LIN {X 0,Y 367.219,Z 542.125,A -85,B 0,C 180,E1 -12876.018,E2 -12876.018} C_VEL
LIN {X 0,Y 366.921,Z 543.374,A -85,B 0,C 180,E1 -12876.247,E2 -12876.247} C_VEL
LIN {X 0,Y 365.149,Z 553.236,A -85,B 0,C 180,E1 -12878.302,E2 -12878.302} C_VEL
LIN {X 0,Y 363.652,Z 562.404,A -85,B 0,C 180,E1 -12880.582,E2 -12880.582} C_VEL
LIN {X 0,Y 362.474,Z 570.103,A -85,B 0,C 180,E1 -12882.886,E2 -12882.886} C_VEL
LIN {X 0,Y 361.538,Z 576.427,A -85,B 0,C 180,E1 -12885.216,E2 -12885.216} C_VEL
LIN {X 0,Y 360.968,Z 581.274,A -85,B 0,C 180,E1 -12887.439,E2 -12887.439} C_VEL
LIN {X 0,Y 360.588,Z 584.605,A -85,B 0,C 180,E1 -12889.352,E2 -12889.352} C_VEL
LIN {X 0,Y 360.218,Z 587.726,A -85,B 0,C 180,E1 -12891.761,E2 -12891.761} C_VEL
LIN {X 0,Y 360.039,Z 589.765,A -85,B 0,C 180,E1 -12894.202,E2 -12894.202} C_VEL
LIN {X 0,Y 360.038,Z 590.58,A -85,B 0,C 180,E1 -12896.679,E2 -12896.679} C_VEL
LIN {X 0,Y 360.098,Z 590.255,A -85,B 0,C 180,E1 -12899.206,E2 -12899.206} C_VEL
LIN {X 0,Y 360.219,Z 588.701,A -85,B 0,C 180,E1 -12901.79,E2 -12901.79} C_VEL
LIN {X 0,Y 360.383,Z 587.415,A -85,B 0,C 180,E1 -12903.098,E2 -12903.098} C_VEL
LIN {X 0,Y 360.836,Z 583.71,A -85,B 0,C 180,E1 -12905.756,E2 -12905.756} C_VEL
LIN {X 0,Y 361.537,Z 578.446,A -85,B 0,C 180,E1 -12908.468,E2 -12908.468} C_VEL
LIN {X 0,Y 362.453,Z 572.426,A -85,B 0,C 180,E1 -12910.868,E2 -12910.868} C_VEL
LIN {X 0,Y 363.696,Z 564.839,A -85,B 0,C 180,E1 -12913.315,E2 -12913.315} C_VEL
LIN {X 0,Y 365.109,Z 556.956,A -85,B 0,C 180,E1 -12915.417,E2 -12915.417} C_VEL
LIN {X 0,Y 366.958,Z 547.569,A -85,B 0,C 180,E1 -12917.508,E2 -12917.508} C_VEL
LIN {X 0,Y 369.193,Z 536.056,A -85,B 0,C 180,E1 -12919.666,E2 -12919.666} C_VEL
LIN {X 0,Y 371.386,Z 524.57,A -85,B 0,C 180,E1 -12921.48,E2 -12921.48} C_VEL
LIN {X 0,Y 373.724,Z 512.125,A -85,B 0,C 180,E1 -12923.14,E2 -12923.14} C_VEL
LIN {X 0,Y 376.004,Z 499.108,A -85,B 0,C 180,E1 -12924.589,E2 -12924.589} C_VEL
LIN {X 0,Y 378.24,Z 484.852,A -85,B 0,C 180,E1 -12925.921,E2 -12925.921} C_VEL
LIN {X 0,Y 380.349,Z 469.499,A -85,B 0,C 180,E1 -12927.097,E2 -12927.097} C_VEL
LIN {X 0,Y 382.181,Z 454.471,A -85,B 0,C 180,E1 -12928.018,E2 -12928.018} C_VEL
LIN {X 0,Y 383.744,Z 437.956,A -85,B 0,C 180,E1 -12928.798,E2 -12928.798} C_VEL
LIN {X 0,Y 384.867,Z 421.878,A -85,B 0,C 180,E1 -12929.343,E2 -12929.343} C_VEL
LIN {X 0,Y 385.749,Z 399.249,A -85,B 0,C 180,E1 -12929.848,E2 -12929.848} C_VEL
LIN {X 0,Y 390.453,Z 263.095,A -85,B 0,C 180,E1 -12932.539,E2 -12932.539} C_VEL
LIN {X 0,Y 382.124,Z 246.592,A -85,B 0,C 180,E1 -12933.936,E2 -12933.936} C_VEL
LIN {X 0,Y 375.065,Z 234.123,A -85,B 0,C 180,E1 -12935.165,E2 -12935.165} C_VEL
LIN {X 0,Y 367.961,Z 222.595,A -85,B 0,C 180,E1 -12936.463,E2 -12936.463} C_VEL
LIN {X 0,Y 365.004,Z 218.068,A -85,B 0,C 180,E1 -12937.021,E2 -12937.021} C_VEL
LIN {X 0,Y 362.52,Z 214.897,A -85,B 0,C 180,E1 -12937.487,E2 -12937.487} C_VEL
LIN {X 0,Y 362.058,Z 213.583,A -85,B 0,C 180,E1 -12937.607,E2 -12937.607} C_VEL
LIN {X 0,Y 361.885,Z 212.725,A -85,B 0,C 180,E1 -12937.821,E2 -12937.821} C_VEL
LIN {X 0,Y 361.961,Z 212.701,A -85,B 0,C 180,E1 -12941.9,E2 -12941.9} C_VEL
LIN {X 0,Y 361.966,Z 212.707,A -85,B 0,C 180,E1 -12945.379,E2 -12945.379} C_VEL
LIN {X 0,Y 361.973,Z 212.708,A -85,B 0,C 180,E1 -12948.804,E2 -12948.804} C_VEL
LIN {X 0,Y 362.119,Z 212.69,A -85,B 0,C 180,E1 -12952.191,E2 -12952.191} C_VEL
LIN {X 0,Y 362.116,Z 212.689,A -85,B 0,C 180,E1 -12954.431,E2 -12954.431} C_VEL
LIN {X 0,Y 362.28,Z 212.673,A -85,B 0,C 180,E1 -12957.776,E2 -12957.776} C_VEL
LIN {X 0,Y 362.406,Z 212.656,A -85,B 0,C 180,E1 -12959.999,E2 -12959.999} C_VEL
LIN {X 0,Y 362.281,Z 212.668,A -85,B 0,C 180,E1 -12962.223,E2 -12962.223} C_VEL
LIN {X 0,Y 362.148,Z 212.685,A -85,B 0,C 180,E1 -12966.686,E2 -12966.686} C_VEL
LIN {X 0,Y 362.001,Z 212.699,A -85,B 0,C 180,E1 -12970.062,E2 -12970.062} C_VEL
LIN {X 0,Y 362,Z 212.704,A -85,B 0,C 180,E1 -12973.898,E2 -12973.898} C_VEL
LIN {X 0,Y 361.929,Z 212.711,A -85,B 0,C 180,E1 -12976.934,E2 -12976.934} C_VEL
LIN {X 0,Y 361.885,Z 212.719,A -85,B 0,C 180,E1 -12980.46,E2 -12980.46} C_VEL
LIN {X 0,Y 361.896,Z 212.713,A -85,B 0,C 180,E1 -12984.112,E2 -12984.112} C_VEL
LIN {X 0,Y 361.943,Z 212.709,A -85,B 0,C 180,E1 -12986.72,E2 -12986.72} C_VEL
LIN {X 0,Y 361.866,Z 212.72,A -85,B 0,C 180,E1 -12990.328,E2 -12990.328} C_VEL
LIN {X 0,Y 361.855,Z 212.719,A -85,B 0,C 180,E1 -12994.28,E2 -12994.28} C_VEL
LIN {X 0,Y 361.864,Z 212.723,A -85,B 0,C 180,E1 -12997.222,E2 -12997.222} C_VEL
LIN {X 0,Y 361.831,Z 212.716,A -85,B 0,C 180,E1 -13000.753,E2 -13000.753} C_VEL
LIN {X 0,Y 361.817,Z 212.721,A -85,B 0,C 180,E1 -13004.368,E2 -13004.368} C_VEL
LIN {X 0,Y 361.851,Z 212.759,A -85,B 0,C 180,E1 -13006.761,E2 -13006.761} C_VEL
LIN {X 0,Y 367.533,Z 227.613,A -85,B 0,C 180,E1 -13010.242,E2 -13010.242} C_VEL
LIN {X 0,Y 376.424,Z 243.115,A -85,B 0,C 180,E1 -13011.885,E2 -13011.885} C_VEL
LIN {X 0,Y 383.341,Z 256.26,A -85,B 0,C 180,E1 -13013.092,E2 -13013.092} C_VEL
LIN {X 0,Y 389.462,Z 269.123,A -85,B 0,C 180,E1 -13014.13,E2 -13014.13} C_VEL
LIN {X 0,Y 390.227,Z 274.285,A -85,B 0,C 180,E1 -13014.34,E2 -13014.34} C_VEL
LIN {X 0,Y 384.653,Z 436.559,A -85,B 0,C 180,E1 -13017.573,E2 -13017.573} C_VEL
LIN {X 0,Y 383.367,Z 452.919,A -85,B 0,C 180,E1 -13018.076,E2 -13018.076} C_VEL
LIN {X 0,Y 381.787,Z 468.385,A -85,B 0,C 180,E1 -13018.741,E2 -13018.741} C_VEL
LIN {X 0,Y 380.071,Z 483.377,A -85,B 0,C 180,E1 -13019.587,E2 -13019.587} C_VEL
LIN {X 0,Y 377.947,Z 498.249,A -85,B 0,C 180,E1 -13020.628,E2 -13020.628} C_VEL
LIN {X 0,Y 375.867,Z 511.427,A -85,B 0,C 180,E1 -13021.761,E2 -13021.761} C_VEL
LIN {X 0,Y 373.487,Z 525.086,A -85,B 0,C 180,E1 -13023.151,E2 -13023.151} C_VEL
LIN {X 0,Y 371.05,Z 538.425,A -85,B 0,C 180,E1 -13024.773,E2 -13024.773} C_VEL
LIN {X 0,Y 368.668,Z 551.545,A -85,B 0,C 180,E1 -13026.697,E2 -13026.697} C_VEL
LIN {X 0,Y 366.53,Z 562.654,A -85,B 0,C 180,E1 -13028.633,E2 -13028.633} C_VEL
LIN {X 0,Y 364.626,Z 573.2,A -85,B 0,C 180,E1 -13030.812,E2 -13030.812} C_VEL
LIN {X 0,Y 363.1,Z 582.538,A -85,B 0,C 180,E1 -13033.12,E2 -13033.12} C_VEL
LIN {X 0,Y 361.972,Z 590.178,A -85,B 0,C 180,E1 -13035.378,E2 -13035.378} C_VEL
LIN {X 0,Y 361.188,Z 596.418,A -85,B 0,C 180,E1 -13037.639,E2 -13037.639} C_VEL
LIN {X 0,Y 360.622,Z 601.516,A -85,B 0,C 180,E1 -13039.896,E2 -13039.896} C_VEL
LIN {X 0,Y 360.448,Z 605.517,A -85,B 0,C 180,E1 -13042.153,E2 -13042.153} C_VEL
LIN {X 0,Y 360.321,Z 608.437,A -85,B 0,C 180,E1 -13044.401,E2 -13044.401} C_VEL
LIN {X 0,Y 360.27,Z 610.381,A -85,B 0,C 180,E1 -13046.642,E2 -13046.642} C_VEL
LIN {X 0,Y 360.318,Z 611.296,A -85,B 0,C 180,E1 -13048.88,E2 -13048.88} C_VEL
LIN {X 0,Y 360.32,Z 611.276,A -85,B 0,C 180,E1 -13051.115,E2 -13051.115} C_VEL
LIN {X 0,Y 360.269,Z 610.225,A -85,B 0,C 180,E1 -13053.352,E2 -13053.352} C_VEL
LIN {X 0,Y 360.373,Z 607.805,A -85,B 0,C 180,E1 -13055.959,E2 -13055.959} C_VEL
LIN {X 0,Y 360.444,Z 605.156,A -85,B 0,C 180,E1 -13057.842,E2 -13057.842} C_VEL
LIN {X 0,Y 360.616,Z 601.081,A -85,B 0,C 180,E1 -13060.099,E2 -13060.099} C_VEL
LIN {X 0,Y 361.38,Z 594.327,A -85,B 0,C 180,E1 -13062.92,E2 -13062.92} C_VEL
LIN {X 0,Y 362.424,Z 585.587,A -85,B 0,C 180,E1 -13065.749,E2 -13065.749} C_VEL
LIN {X 0,Y 363.753,Z 576.983,A -85,B 0,C 180,E1 -13068.003,E2 -13068.003} C_VEL
LIN {X 0,Y 365.114,Z 568.067,A -85,B 0,C 180,E1 -13069.975,E2 -13069.975} C_VEL
LIN {X 0,Y 366.921,Z 557.712,A -85,B 0,C 180,E1 -13071.928,E2 -13071.928} C_VEL
LIN {X 0,Y 368.887,Z 546.364,A -85,B 0,C 180,E1 -13073.746,E2 -13073.746} C_VEL
LIN {X 0,Y 370.776,Z 535.379,A -85,B 0,C 180,E1 -13075.241,E2 -13075.241} C_VEL
LIN {X 0,Y 372.93,Z 522.597,A -85,B 0,C 180,E1 -13076.735,E2 -13076.735} C_VEL
LIN {X 0,Y 375.092,Z 508.802,A -85,B 0,C 180,E1 -13078.087,E2 -13078.087} C_VEL
LIN {X 0,Y 377.203,Z 494.008,A -85,B 0,C 180,E1 -13079.276,E2 -13079.276} C_VEL
LIN {X 0,Y 379.094,Z 478.909,A -85,B 0,C 180,E1 -13080.263,E2 -13080.263} C_VEL
LIN {X 0,Y 380.72,Z 463.094,A -85,B 0,C 180,E1 -13081.08,E2 -13081.08} C_VEL
LIN {X 0,Y 382.112,Z 447.18,A -85,B 0,C 180,E1 -13081.686,E2 -13081.686} C_VEL
LIN {X 0,Y 383.114,Z 429.543,A -85,B 0,C 180,E1 -13082.135,E2 -13082.135} C_VEL
LIN {X 0,Y 387.859,Z 273.803,A -85,B 0,C 180,E1 -13085.17,E2 -13085.17} C_VEL
LIN {X 0,Y 386.671,Z 267.24,A -85,B 0,C 180,E1 -13085.435,E2 -13085.435} C_VEL
LIN {X 0,Y 376.6,Z 246.193,A -85,B 0,C 180,E1 -13086.955,E2 -13086.955} C_VEL
LIN {X 0,Y 367.525,Z 229.148,A -85,B 0,C 180,E1 -13088.37,E2 -13088.37} C_VEL
LIN {X 0,Y 363.515,Z 217.682,A -85,B 0,C 180,E1 -13090.639,E2 -13090.639} C_VEL
LIN {X 0,Y 361.829,Z 212.725,A -85,B 0,C 180,E1 -13091.693,E2 -13091.693} C_VEL
LIN {X 0,Y 361.801,Z 212.72,A -85,B 0,C 180,E1 -13095.63,E2 -13095.63} C_VEL
LIN {X 0,Y 361.849,Z 212.713,A -85,B 0,C 180,E1 -13099.235,E2 -13099.235} C_VEL
LIN {X 0,Y 361.844,Z 212.712,A -85,B 0,C 180,E1 -13102.98,E2 -13102.98} C_VEL
LIN {X 0,Y 361.832,Z 212.721,A -85,B 0,C 180,E1 -13106.629,E2 -13106.629} C_VEL
LIN {X 0,Y 361.837,Z 212.723,A -85,B 0,C 180,E1 -13109.669,E2 -13109.669} C_VEL
LIN {X 0,Y 361.925,Z 212.693,A -85,B 0,C 180,E1 -13113.473,E2 -13113.473} C_VEL
LIN {X 0,Y 361.88,Z 212.722,A -85,B 0,C 180,E1 -13117.145,E2 -13117.145} C_VEL
LIN {X 0,Y 361.903,Z 212.692,A -85,B 0,C 180,E1 -13120.724,E2 -13120.724} C_VEL
LIN {X 0,Y 361.916,Z 212.715,A -85,B 0,C 180,E1 -13124.225,E2 -13124.225} C_VEL
LIN {X 0,Y 361.969,Z 212.684,A -85,B 0,C 180,E1 -13126.527,E2 -13126.527} C_VEL
LIN {X 0,Y 362.005,Z 212.694,A -85,B 0,C 180,E1 -13129.938,E2 -13129.938} C_VEL
LIN {X 0,Y 362.138,Z 212.681,A -85,B 0,C 180,E1 -13133.314,E2 -13133.314} C_VEL
LIN {X 0,Y 362.251,Z 212.65,A -85,B 0,C 180,E1 -13137.777,E2 -13137.777} C_VEL
LIN {X 0,Y 362.398,Z 212.651,A -85,B 0,C 180,E1 -13140.001,E2 -13140.001} C_VEL
LIN {X 0,Y 362.251,Z 212.673,A -85,B 0,C 180,E1 -13142.224,E2 -13142.224} C_VEL
LIN {X 0,Y 362.132,Z 212.682,A -85,B 0,C 180,E1 -13146.687,E2 -13146.687} C_VEL
LIN {X 0,Y 362.001,Z 212.695,A -85,B 0,C 180,E1 -13150.063,E2 -13150.063} C_VEL
LIN {X 0,Y 361.969,Z 212.7,A -85,B 0,C 180,E1 -13153.9,E2 -13153.9} C_VEL
LIN {X 0,Y 361.94,Z 212.696,A -85,B 0,C 180,E1 -13157.941,E2 -13157.941} C_VEL
LIN {X 0,Y 361.866,Z 212.717,A -85,B 0,C 180,E1 -13161.655,E2 -13161.655} C_VEL
LIN {X 0,Y 361.903,Z 212.699,A -85,B 0,C 180,E1 -13165.293,E2 -13165.293} C_VEL
LIN {X 0,Y 361.889,Z 212.71,A -85,B 0,C 180,E1 -13167.781,E2 -13167.781} C_VEL
LIN {X 0,Y 361.824,Z 212.719,A -85,B 0,C 180,E1 -13171.288,E2 -13171.288} C_VEL
LIN {X 0,Y 361.832,Z 212.715,A -85,B 0,C 180,E1 -13174.284,E2 -13174.284} C_VEL
LIN {X 0,Y 361.842,Z 212.721,A -85,B 0,C 180,E1 -13177.226,E2 -13177.226} C_VEL
LIN {X 0,Y 361.816,Z 212.722,A -85,B 0,C 180,E1 -13180.758,E2 -13180.758} C_VEL
LIN {X 0,Y 361.799,Z 212.716,A -85,B 0,C 180,E1 -13184.372,E2 -13184.372} C_VEL
LIN {X 0,Y 361.818,Z 212.727,A -85,B 0,C 180,E1 -13187.572,E2 -13187.572} C_VEL
LIN {X 0,Y 361.82,Z 212.716,A -85,B 0,C 180,E1 -13190.984,E2 -13190.984} C_VEL
LIN {X 0,Y 361.863,Z 212.712,A -85,B 0,C 180,E1 -13194.659,E2 -13194.659} C_VEL
LIN {X 0,Y 361.829,Z 212.726,A -85,B 0,C 180,E1 -13198.374,E2 -13198.374} C_VEL
LIN {X 0,Y 361.858,Z 212.718,A -85,B 0,C 180,E1 -13200.956,E2 -13200.956} C_VEL
LIN {X 0,Y 361.877,Z 212.714,A -85,B 0,C 180,E1 -13204.71,E2 -13204.71} C_VEL
LIN {X 0,Y 361.851,Z 212.72,A -85,B 0,C 180,E1 -13208.348,E2 -13208.348} C_VEL
LIN {X 0,Y 361.918,Z 212.72,A -85,B 0,C 180,E1 -13212.088,E2 -13212.088} C_VEL
LIN {X 0,Y 361.981,Z 212.704,A -85,B 0,C 180,E1 -13216.115,E2 -13216.115} C_VEL
LIN {X 0,Y 361.956,Z 212.707,A -85,B 0,C 180,E1 -13218.055,E2 -13218.055} C_VEL
LIN {X 0,Y 362.948,Z 215.516,A -85,B 0,C 180,E1 -13218.254,E2 -13218.254} C_VEL
LIN {X 0,Y 364.51,Z 217.644,A -85,B 0,C 180,E1 -13218.491,E2 -13218.491} C_VEL
LIN {X 0,Y 373.334,Z 232.468,A -85,B 0,C 180,E1 -13219.859,E2 -13219.859} C_VEL
LIN {X 0,Y 381.122,Z 247.442,A -85,B 0,C 180,E1 -13221.038,E2 -13221.038} C_VEL
LIN {X 0,Y 387.956,Z 261.424,A -85,B 0,C 180,E1 -13222.048,E2 -13222.048} C_VEL
LIN {X 0,Y 383.102,Z 417.262,A -85,B 0,C 180,E1 -13225.103,E2 -13225.103} C_VEL
LIN {X 0,Y 382.07,Z 433.744,A -85,B 0,C 180,E1 -13225.618,E2 -13225.618} C_VEL
LIN {X 0,Y 380.73,Z 449.833,A -85,B 0,C 180,E1 -13226.328,E2 -13226.328} C_VEL
LIN {X 0,Y 379.108,Z 465.262,A -85,B 0,C 180,E1 -13227.213,E2 -13227.213} C_VEL
LIN {X 0,Y 377.356,Z 479.93,A -85,B 0,C 180,E1 -13228.268,E2 -13228.268} C_VEL
LIN {X 0,Y 375.115,Z 495.059,A -85,B 0,C 180,E1 -13229.6,E2 -13229.6} C_VEL
LIN {X 0,Y 372.931,Z 508.887,A -85,B 0,C 180,E1 -13231.082,E2 -13231.082} C_VEL
LIN {X 0,Y 370.628,Z 522.373,A -85,B 0,C 180,E1 -13232.811,E2 -13232.811} C_VEL
LIN {X 0,Y 368.554,Z 534.4,A -85,B 0,C 180,E1 -13234.651,E2 -13234.651} C_VEL
LIN {X 0,Y 366.921,Z 543.374,A -85,B 0,C 180,E1 -13236.247,E2 -13236.247} C_VEL
LIN {X 0,Y 365.622,Z 547.103,A -85,B 0,C 180,E1 -13236.936,E2 -13236.936} C_VEL
LIN {X 0,Y 358.662,Z 557.399,A -85,B 0,C 180,E1 -13238.972,E2 -13238.972} C_VEL
LIN {X 0,Y 357.128,Z 560.591,A -85,B 0,C 180,E1 -13239.732,E2 -13239.732} C_VEL
LIN {X 0,Y 356.889,Z 561.583,A -85,B 0,C 180,E1 -13239.999,E2 -13239.999} C_VEL
LIN {X 0,Y 355.521,Z 570.101,A -85,B 0,C 180,E1 -13242.562,E2 -13242.562} C_VEL
LIN {X 0,Y 354.542,Z 576.449,A -85,B 0,C 180,E1 -13244.936,E2 -13244.936} C_VEL
LIN {X 0,Y 353.873,Z 582.045,A -85,B 0,C 180,E1 -13247.579,E2 -13247.579} C_VEL
LIN {X 0,Y 353.444,Z 585.626,A -85,B 0,C 180,E1 -13249.759,E2 -13249.759} C_VEL
LIN {X 0,Y 353.06,Z 588.471,A -85,B 0,C 180,E1 -13252.225,E2 -13252.225} C_VEL
LIN {X 0,Y 352.933,Z 590.215,A -85,B 0,C 180,E1 -13254.721,E2 -13254.721} C_VEL
LIN {X 0,Y 352.947,Z 590.86,A -85,B 0,C 180,E1 -13257.259,E2 -13257.259} C_VEL
LIN {X 0,Y 353.01,Z 590.23,A -85,B 0,C 180,E1 -13259.851,E2 -13259.851} C_VEL
LIN {X 0,Y 353.196,Z 588.343,A -85,B 0,C 180,E1 -13262.499,E2 -13262.499} C_VEL
LIN {X 0,Y 353.378,Z 586.897,A -85,B 0,C 180,E1 -13263.841,E2 -13263.841} C_VEL
LIN {X 0,Y 353.93,Z 582.903,A -85,B 0,C 180,E1 -13266.565,E2 -13266.565} C_VEL
LIN {X 0,Y 354.518,Z 578.826,A -85,B 0,C 180,E1 -13268.644,E2 -13268.644} C_VEL
LIN {X 0,Y 355.613,Z 572.211,A -85,B 0,C 180,E1 -13271.322,E2 -13271.322} C_VEL
LIN {X 0,Y 357.004,Z 564.09,A -85,B 0,C 180,E1 -13273.939,E2 -13273.939} C_VEL
LIN {X 0,Y 358.628,Z 556.076,A -85,B 0,C 180,E1 -13276.071,E2 -13276.071} C_VEL
LIN {X 0,Y 360.56,Z 546.533,A -85,B 0,C 180,E1 -13278.197,E2 -13278.197} C_VEL
LIN {X 0,Y 362.805,Z 535.508,A -85,B 0,C 180,E1 -13280.263,E2 -13280.263} C_VEL
LIN {X 0,Y 365.158,Z 523.855,A -85,B 0,C 180,E1 -13282.103,E2 -13282.103} C_VEL
LIN {X 0,Y 367.605,Z 511.217,A -85,B 0,C 180,E1 -13283.79,E2 -13283.79} C_VEL
LIN {X 0,Y 369.972,Z 498.095,A -85,B 0,C 180,E1 -13285.257,E2 -13285.257} C_VEL
LIN {X 0,Y 372.295,Z 483.968,A -85,B 0,C 180,E1 -13286.569,E2 -13286.569} C_VEL
LIN {X 0,Y 374.312,Z 469.787,A -85,B 0,C 180,E1 -13287.664,E2 -13287.664} C_VEL
LIN {X 0,Y 376.249,Z 454.47,A -85,B 0,C 180,E1 -13288.613,E2 -13288.613} C_VEL
LIN {X 0,Y 377.877,Z 437.865,A -85,B 0,C 180,E1 -13289.407,E2 -13289.407} C_VEL
LIN {X 0,Y 379.012,Z 422.225,A -85,B 0,C 180,E1 -13289.94,E2 -13289.94} C_VEL
LIN {X 0,Y 379.946,Z 399.352,A -85,B 0,C 180,E1 -13290.458,E2 -13290.458} C_VEL
LIN {X 0,Y 384.734,Z 265.474,A -85,B 0,C 180,E1 -13293.148,E2 -13293.148} C_VEL
LIN {X 0,Y 377.424,Z 250.859,A -85,B 0,C 180,E1 -13294.421,E2 -13294.421} C_VEL
LIN {X 0,Y 370.711,Z 238.798,A -85,B 0,C 180,E1 -13295.635,E2 -13295.635} C_VEL
LIN {X 0,Y 363.511,Z 227.092,A -85,B 0,C 180,E1 -13296.989,E2 -13296.989} C_VEL
LIN {X 0,Y 360.024,Z 222.128,A -85,B 0,C 180,E1 -13297.663,E2 -13297.663} C_VEL
LIN {X 0,Y 357.91,Z 218.725,A -85,B 0,C 180,E1 -13298.093,E2 -13298.093} C_VEL
LIN {X 0,Y 355.666,Z 216.157,A -85,B 0,C 180,E1 -13298.532,E2 -13298.532} C_VEL
LIN {X 0,Y 354.871,Z 213.682,A -85,B 0,C 180,E1 -13298.786,E2 -13298.786} C_VEL
LIN {X 0,Y 354.903,Z 213.577,A -85,B 0,C 180,E1 -13302.719,E2 -13302.719} C_VEL
LIN {X 0,Y 354.955,Z 213.585,A -85,B 0,C 180,E1 -13306.255,E2 -13306.255} C_VEL
LIN {X 0,Y 354.96,Z 213.58,A -85,B 0,C 180,E1 -13309.735,E2 -13309.735} C_VEL
LIN {X 0,Y 355.127,Z 213.563,A -85,B 0,C 180,E1 -13313.18,E2 -13313.18} C_VEL
LIN {X 0,Y 355.244,Z 213.549,A -85,B 0,C 180,E1 -13317.732,E2 -13317.732} C_VEL
LIN {X 0,Y 355.356,Z 213.534,A -85,B 0,C 180,E1 -13319.999,E2 -13319.999} C_VEL
LIN {X 0,Y 355.244,Z 213.544,A -85,B 0,C 180,E1 -13322.267,E2 -13322.267} C_VEL
LIN {X 0,Y 355.112,Z 213.561,A -85,B 0,C 180,E1 -13326.819,E2 -13326.819} C_VEL
LIN {X 0,Y 354.957,Z 213.576,A -85,B 0,C 180,E1 -13330.264,E2 -13330.264} C_VEL
LIN {X 0,Y 354.945,Z 213.584,A -85,B 0,C 180,E1 -13334.018,E2 -13334.018} C_VEL
LIN {X 0,Y 354.892,Z 213.588,A -85,B 0,C 180,E1 -13338.091,E2 -13338.091} C_VEL
LIN {X 0,Y 354.819,Z 213.595,A -85,B 0,C 180,E1 -13342.106,E2 -13342.106} C_VEL
LIN {X 0,Y 354.9,Z 213.59,A -85,B 0,C 180,E1 -13345.827,E2 -13345.827} C_VEL
LIN {X 0,Y 354.816,Z 213.596,A -85,B 0,C 180,E1 -13349.681,E2 -13349.681} C_VEL
LIN {X 0,Y 354.809,Z 213.599,A -85,B 0,C 180,E1 -13353.701,E2 -13353.701} C_VEL
LIN {X 0,Y 354.798,Z 213.599,A -85,B 0,C 180,E1 -13356.459,E2 -13356.459} C_VEL
LIN {X 0,Y 354.827,Z 213.601,A -85,B 0,C 180,E1 -13359.423,E2 -13359.423} C_VEL
LIN {X 0,Y 354.788,Z 213.606,A -85,B 0,C 180,E1 -13362.866,E2 -13362.866} C_VEL
LIN {X 0,Y 354.791,Z 213.658,A -85,B 0,C 180,E1 -13365.749,E2 -13365.749} C_VEL
LIN {X 0,Y 360.099,Z 227.361,A -85,B 0,C 180,E1 -13369.136,E2 -13369.136} C_VEL
LIN {X 0,Y 368.027,Z 240.648,A -85,B 0,C 180,E1 -13370.678,E2 -13370.678} C_VEL
LIN {X 0,Y 376.256,Z 255.76,A -85,B 0,C 180,E1 -13372.192,E2 -13372.192} C_VEL
LIN {X 0,Y 384.055,Z 271.958,A -85,B 0,C 180,E1 -13373.567,E2 -13373.567} C_VEL
LIN {X 0,Y 384.577,Z 275.959,A -85,B 0,C 180,E1 -13373.727,E2 -13373.727} C_VEL
LIN {X 0,Y 378.828,Z 436.068,A -85,B 0,C 180,E1 -13376.962,E2 -13376.962} C_VEL
LIN {X 0,Y 377.476,Z 452.712,A -85,B 0,C 180,E1 -13377.478,E2 -13377.478} C_VEL
LIN {X 0,Y 375.753,Z 468.781,A -85,B 0,C 180,E1 -13378.181,E2 -13378.181} C_VEL
LIN {X 0,Y 373.685,Z 485.569,A -85,B 0,C 180,E1 -13379.168,E2 -13379.168} C_VEL
LIN {X 0,Y 371.507,Z 500.008,A -85,B 0,C 180,E1 -13380.224,E2 -13380.224} C_VEL
LIN {X 0,Y 368.991,Z 514.956,A -85,B 0,C 180,E1 -13381.563,E2 -13381.563} C_VEL
LIN {X 0,Y 366.447,Z 528.64,A -85,B 0,C 180,E1 -13383.056,E2 -13383.056} C_VEL
LIN {X 0,Y 364.19,Z 540.37,A -85,B 0,C 180,E1 -13384.57,E2 -13384.57} C_VEL
LIN {X 0,Y 362.077,Z 551.511,A -85,B 0,C 180,E1 -13386.247,E2 -13386.247} C_VEL
LIN {X 0,Y 359.836,Z 562.578,A -85,B 0,C 180,E1 -13388.215,E2 -13388.215} C_VEL
LIN {X 0,Y 358.024,Z 572.093,A -85,B 0,C 180,E1 -13390.205,E2 -13390.205} C_VEL
LIN {X 0,Y 356.415,Z 581.386,A -85,B 0,C 180,E1 -13392.498,E2 -13392.498} C_VEL
LIN {X 0,Y 355.004,Z 590.035,A -85,B 0,C 180,E1 -13395.084,E2 -13395.084} C_VEL
LIN {X 0,Y 354.184,Z 596.269,A -85,B 0,C 180,E1 -13397.39,E2 -13397.39} C_VEL
LIN {X 0,Y 353.569,Z 601.352,A -85,B 0,C 180,E1 -13399.692,E2 -13399.692} C_VEL
LIN {X 0,Y 353.359,Z 605.343,A -85,B 0,C 180,E1 -13401.995,E2 -13401.995} C_VEL
LIN {X 0,Y 353.239,Z 608.25,A -85,B 0,C 180,E1 -13404.288,E2 -13404.288} C_VEL
LIN {X 0,Y 353.191,Z 610.19,A -85,B 0,C 180,E1 -13406.575,E2 -13406.575} C_VEL
LIN {X 0,Y 353.218,Z 611.093,A -85,B 0,C 180,E1 -13408.857,E2 -13408.857} C_VEL
LIN {X 0,Y 353.221,Z 611.068,A -85,B 0,C 180,E1 -13411.137,E2 -13411.137} C_VEL
LIN {X 0,Y 353.19,Z 610.004,A -85,B 0,C 180,E1 -13413.419,E2 -13413.419} C_VEL
LIN {X 0,Y 353.272,Z 607.792,A -85,B 0,C 180,E1 -13415.905,E2 -13415.905} C_VEL
LIN {X 0,Y 353.355,Z 604.913,A -85,B 0,C 180,E1 -13418,E2 -13418} C_VEL
LIN {X 0,Y 353.553,Z 600.825,A -85,B 0,C 180,E1 -13420.303,E2 -13420.303} C_VEL
LIN {X 0,Y 354.361,Z 594.051,A -85,B 0,C 180,E1 -13423.181,E2 -13423.181} C_VEL
LIN {X 0,Y 355.182,Z 587.17,A -85,B 0,C 180,E1 -13425.49,E2 -13425.49} C_VEL
LIN {X 0,Y 356.523,Z 578.922,A -85,B 0,C 180,E1 -13427.787,E2 -13427.787} C_VEL
LIN {X 0,Y 357.864,Z 570.444,A -85,B 0,C 180,E1 -13429.798,E2 -13429.798} C_VEL
LIN {X 0,Y 359.656,Z 560.442,A -85,B 0,C 180,E1 -13431.791,E2 -13431.791} C_VEL
LIN {X 0,Y 361.794,Z 548.753,A -85,B 0,C 180,E1 -13433.767,E2 -13433.767} C_VEL
LIN {X 0,Y 363.847,Z 537.071,A -85,B 0,C 180,E1 -13435.449,E2 -13435.449} C_VEL
LIN {X 0,Y 366.287,Z 523.374,A -85,B 0,C 180,E1 -13437.105,E2 -13437.105} C_VEL
LIN {X 0,Y 368.522,Z 509.751,A -85,B 0,C 180,E1 -13438.47,E2 -13438.47} C_VEL
LIN {X 0,Y 370.698,Z 495.143,A -85,B 0,C 180,E1 -13439.685,E2 -13439.685} C_VEL
LIN {X 0,Y 372.787,Z 479.278,A -85,B 0,C 180,E1 -13440.751,E2 -13440.751} C_VEL
LIN {X 0,Y 374.471,Z 463.663,A -85,B 0,C 180,E1 -13441.579,E2 -13441.579} C_VEL
LIN {X 0,Y 375.974,Z 446.995,A -85,B 0,C 180,E1 -13442.226,E2 -13442.226} C_VEL
LIN {X 0,Y 377.008,Z 429.378,A -85,B 0,C 180,E1 -13442.681,E2 -13442.681} C_VEL
LIN {X 0,Y 381.873,Z 274.132,A -85,B 0,C 180,E1 -13445.757,E2 -13445.757} C_VEL
LIN {X 0,Y 381.018,Z 270.109,A -85,B 0,C 180,E1 -13445.936,E2 -13445.936} C_VEL
LIN {X 0,Y 371.199,Z 249.636,A -85,B 0,C 180,E1 -13447.455,E2 -13447.455} C_VEL
LIN {X 0,Y 361.504,Z 231.441,A -85,B 0,C 180,E1 -13449.007,E2 -13449.007} C_VEL
LIN {X 0,Y 360.206,Z 228.75,A -85,B 0,C 180,E1 -13449.255,E2 -13449.255} C_VEL
LIN {X 0,Y 354.794,Z 213.594,A -85,B 0,C 180,E1 -13452.43,E2 -13452.43} C_VEL
LIN {X 0,Y 354.754,Z 213.599,A -85,B 0,C 180,E1 -13456.102,E2 -13456.102} C_VEL
LIN {X 0,Y 354.801,Z 213.591,A -85,B 0,C 180,E1 -13459.182,E2 -13459.182} C_VEL
LIN {X 0,Y 354.785,Z 213.596,A -85,B 0,C 180,E1 -13462.4,E2 -13462.4} C_VEL
LIN {X 0,Y 354.787,Z 213.6,A -85,B 0,C 180,E1 -13464.939,E2 -13464.939} C_VEL
LIN {X 0,Y 354.766,Z 213.587,A -85,B 0,C 180,E1 -13468.403,E2 -13468.403} C_VEL
LIN {X 0,Y 354.819,Z 213.598,A -85,B 0,C 180,E1 -13471.617,E2 -13471.617} C_VEL
LIN {X 0,Y 354.871,Z 213.572,A -85,B 0,C 180,E1 -13474.171,E2 -13474.171} C_VEL
LIN {X 0,Y 354.825,Z 213.596,A -85,B 0,C 180,E1 -13477.894,E2 -13477.894} C_VEL
LIN {X 0,Y 354.894,Z 213.58,A -85,B 0,C 180,E1 -13481.89,E2 -13481.89} C_VEL
LIN {X 0,Y 354.913,Z 213.573,A -85,B 0,C 180,E1 -13485.981,E2 -13485.981} C_VEL
LIN {X 0,Y 354.952,Z 213.572,A -85,B 0,C 180,E1 -13489.736,E2 -13489.736} C_VEL
LIN {X 0,Y 355.101,Z 213.558,A -85,B 0,C 180,E1 -13493.181,E2 -13493.181} C_VEL
LIN {X 0,Y 355.215,Z 213.524,A -85,B 0,C 180,E1 -13497.733,E2 -13497.733} C_VEL
LIN {X 0,Y 355.367,Z 213.527,A -85,B 0,C 180,E1 -13500.001,E2 -13500.001} C_VEL
LIN {X 0,Y 355.214,Z 213.548,A -85,B 0,C 180,E1 -13502.268,E2 -13502.268} C_VEL
LIN {X 0,Y 355.096,Z 213.56,A -85,B 0,C 180,E1 -13506.821,E2 -13506.821} C_VEL
LIN {X 0,Y 354.948,Z 213.569,A -85,B 0,C 180,E1 -13510.266,E2 -13510.266} C_VEL
LIN {X 0,Y 354.914,Z 213.58,A -85,B 0,C 180,E1 -13514.02,E2 -13514.02} C_VEL
LIN {X 0,Y 354.895,Z 213.571,A -85,B 0,C 180,E1 -13518.11,E2 -13518.11} C_VEL
LIN {X 0,Y 354.808,Z 213.599,A -85,B 0,C 180,E1 -13522.108,E2 -13522.108} C_VEL
LIN {X 0,Y 354.874,Z 213.571,A -85,B 0,C 180,E1 -13525.83,E2 -13525.83} C_VEL
LIN {X 0,Y 354.831,Z 213.597,A -85,B 0,C 180,E1 -13529.681,E2 -13529.681} C_VEL
LIN {X 0,Y 354.785,Z 213.587,A -85,B 0,C 180,E1 -13533.705,E2 -13533.705} C_VEL
LIN {X 0,Y 354.777,Z 213.605,A -85,B 0,C 180,E1 -13536.463,E2 -13536.463} C_VEL
LIN {X 0,Y 354.806,Z 213.58,A -85,B 0,C 180,E1 -13539.427,E2 -13539.427} C_VEL
LIN {X 0,Y 354.771,Z 213.604,A -85,B 0,C 180,E1 -13542.871,E2 -13542.871} C_VEL
LIN {X 0,Y 354.75,Z 213.595,A -85,B 0,C 180,E1 -13546.107,E2 -13546.107} C_VEL
LIN {X 0,Y 354.769,Z 213.601,A -85,B 0,C 180,E1 -13549.182,E2 -13549.182} C_VEL
LIN {X 0,Y 354.79,Z 213.604,A -85,B 0,C 180,E1 -13552.407,E2 -13552.407} C_VEL
LIN {X 0,Y 354.801,Z 213.59,A -85,B 0,C 180,E1 -13554.944,E2 -13554.944} C_VEL
LIN {X 0,Y 354.784,Z 213.603,A -85,B 0,C 180,E1 -13558.409,E2 -13558.409} C_VEL
LIN {X 0,Y 354.794,Z 213.601,A -85,B 0,C 180,E1 -13561.618,E2 -13561.618} C_VEL
LIN {X 0,Y 354.829,Z 213.598,A -85,B 0,C 180,E1 -13565.661,E2 -13565.661} C_VEL
LIN {X 0,Y 354.823,Z 213.6,A -85,B 0,C 180,E1 -13569.117,E2 -13569.117} C_VEL
LIN {X 0,Y 354.858,Z 213.596,A -85,B 0,C 180,E1 -13572.721,E2 -13572.721} C_VEL
LIN {X 0,Y 354.94,Z 213.581,A -85,B 0,C 180,E1 -13576.258,E2 -13576.258} C_VEL
LIN {X 0,Y 354.961,Z 213.76,A -85,B 0,C 180,E1 -13577.242,E2 -13577.242} C_VEL
LIN {X 0,Y 355.953,Z 216.498,A -85,B 0,C 180,E1 -13577.437,E2 -13577.437} C_VEL
LIN {X 0,Y 357.579,Z 218.773,A -85,B 0,C 180,E1 -13577.695,E2 -13577.695} C_VEL
LIN {X 0,Y 367.054,Z 234.219,A -85,B 0,C 180,E1 -13579.2,E2 -13579.2} C_VEL
LIN {X 0,Y 375.712,Z 250.759,A -85,B 0,C 180,E1 -13580.553,E2 -13580.553} C_VEL
LIN {X 0,Y 381.978,Z 263.827,A -85,B 0,C 180,E1 -13581.505,E2 -13581.505} C_VEL
LIN {X 0,Y 376.992,Z 417.214,A -85,B 0,C 180,E1 -13584.554,E2 -13584.554} C_VEL
LIN {X 0,Y 375.948,Z 433.742,A -85,B 0,C 180,E1 -13585.076,E2 -13585.076} C_VEL
LIN {X 0,Y 374.582,Z 449.425,A -85,B 0,C 180,E1 -13585.77,E2 -13585.77} C_VEL
LIN {X 0,Y 372.949,Z 464.672,A -85,B 0,C 180,E1 -13586.647,E2 -13586.647} C_VEL
LIN {X 0,Y 371.166,Z 479.177,A -85,B 0,C 180,E1 -13587.697,E2 -13587.697} C_VEL
LIN {X 0,Y 368.825,Z 494.489,A -85,B 0,C 180,E1 -13589.047,E2 -13589.047} C_VEL
LIN {X 0,Y 366.784,Z 507.257,A -85,B 0,C 180,E1 -13590.414,E2 -13590.414} C_VEL
LIN {X 0,Y 364.456,Z 520.313,A -85,B 0,C 180,E1 -13592.061,E2 -13592.061} C_VEL
LIN {X 0,Y 362.274,Z 532.519,A -85,B 0,C 180,E1 -13593.896,E2 -13593.896} C_VEL
LIN {X 0,Y 360.071,Z 544.146,A -85,B 0,C 180,E1 -13595.985,E2 -13595.985} C_VEL
LIN {X 0,Y 358.402,Z 553.105,A -85,B 0,C 180,E1 -13597.892,E2 -13597.892} C_VEL
LIN {X 0,Y 356.889,Z 561.583,A -85,B 0,C 180,E1 -13599.999,E2 -13599.999} C_VEL
LIN {X 0,Y 355.792,Z 564.575,A -85,B 0,C 180,E1 -13600.799,E2 -13600.799} C_VEL
LIN {X 0,Y 352.284,Z 569.204,A -85,B 0,C 180,E1 -13602.098,E2 -13602.098} C_VEL
LIN {X 0,Y 348.776,Z 573.417,A -85,B 0,C 180,E1 -13603.456,E2 -13603.456} C_VEL
LIN {X 0,Y 347.703,Z 575.711,A -85,B 0,C 180,E1 -13604.337,E2 -13604.337} C_VEL
LIN {X 0,Y 347.021,Z 580.496,A -85,B 0,C 180,E1 -13606.473,E2 -13606.473} C_VEL
LIN {X 0,Y 346.501,Z 584.77,A -85,B 0,C 180,E1 -13608.939,E2 -13608.939} C_VEL
LIN {X 0,Y 346.078,Z 587.981,A -85,B 0,C 180,E1 -13611.443,E2 -13611.443} C_VEL
LIN {X 0,Y 345.853,Z 590.068,A -85,B 0,C 180,E1 -13613.982,E2 -13613.982} C_VEL
LIN {X 0,Y 345.856,Z 590.974,A -85,B 0,C 180,E1 -13616.604,E2 -13616.604} C_VEL
LIN {X 0,Y 345.905,Z 590.733,A -85,B 0,C 180,E1 -13619.187,E2 -13619.187} C_VEL
LIN {X 0,Y 346.043,Z 589.26,A -85,B 0,C 180,E1 -13621.876,E2 -13621.876} C_VEL
LIN {X 0,Y 346.423,Z 586.365,A -85,B 0,C 180,E1 -13624.616,E2 -13624.616} C_VEL
LIN {X 0,Y 347.087,Z 582,A -85,B 0,C 180,E1 -13627.408,E2 -13627.408} C_VEL
LIN {X 0,Y 347.894,Z 576.936,A -85,B 0,C 180,E1 -13629.855,E2 -13629.855} C_VEL
LIN {X 0,Y 349.076,Z 570.285,A -85,B 0,C 180,E1 -13632.418,E2 -13632.418} C_VEL
LIN {X 0,Y 350.732,Z 561.76,A -85,B 0,C 180,E1 -13635.052,E2 -13635.052} C_VEL
LIN {X 0,Y 352.804,Z 552.08,A -85,B 0,C 180,E1 -13637.483,E2 -13637.483} C_VEL
LIN {X 0,Y 355.042,Z 541.477,A -85,B 0,C 180,E1 -13639.697,E2 -13639.697} C_VEL
LIN {X 0,Y 357.307,Z 530.929,A -85,B 0,C 180,E1 -13641.555,E2 -13641.555} C_VEL
LIN {X 0,Y 359.937,Z 518.435,A -85,B 0,C 180,E1 -13643.416,E2 -13643.416} C_VEL
LIN {X 0,Y 362.437,Z 505.708,A -85,B 0,C 180,E1 -13645.013,E2 -13645.013} C_VEL
LIN {X 0,Y 364.865,Z 492.261,A -85,B 0,C 180,E1 -13646.418,E2 -13646.418} C_VEL
LIN {X 0,Y 367.17,Z 477.98,A -85,B 0,C 180,E1 -13647.662,E2 -13647.662} C_VEL
LIN {X 0,Y 369.188,Z 464.142,A -85,B 0,C 180,E1 -13648.653,E2 -13648.653} C_VEL
LIN {X 0,Y 370.997,Z 448.499,A -85,B 0,C 180,E1 -13649.544,E2 -13649.544} C_VEL
LIN {X 0,Y 372.487,Z 431.923,A -85,B 0,C 180,E1 -13650.258,E2 -13650.258} C_VEL
LIN {X 0,Y 373.597,Z 415.641,A -85,B 0,C 180,E1 -13650.738,E2 -13650.738} C_VEL
LIN {X 0,Y 379.144,Z 267.888,A -85,B 0,C 180,E1 -13653.769,E2 -13653.769} C_VEL
LIN {X 0,Y 372.438,Z 254.553,A -85,B 0,C 180,E1 -13654.978,E2 -13654.978} C_VEL
LIN {X 0,Y 366.342,Z 243.461,A -85,B 0,C 180,E1 -13656.12,E2 -13656.12} C_VEL
LIN {X 0,Y 359.337,Z 231.925,A -85,B 0,C 180,E1 -13657.485,E2 -13657.485} C_VEL
LIN {X 0,Y 355.901,Z 227.09,A -85,B 0,C 180,E1 -13658.166,E2 -13658.166} C_VEL
LIN {X 0,Y 353.368,Z 223.418,A -85,B 0,C 180,E1 -13658.691,E2 -13658.691} C_VEL
LIN {X 0,Y 351.198,Z 220.162,A -85,B 0,C 180,E1 -13659.155,E2 -13659.155} C_VEL
LIN {X 0,Y 350.201,Z 218.969,A -85,B 0,C 180,E1 -13659.362,E2 -13659.362} C_VEL
LIN {X 0,Y 348.393,Z 216.554,A -85,B 0,C 180,E1 -13659.751,E2 -13659.751} C_VEL
LIN {X 0,Y 347.815,Z 214.466,A -85,B 0,C 180,E1 -13659.947,E2 -13659.947} C_VEL
LIN {X 0,Y 347.871,Z 214.452,A -85,B 0,C 180,E1 -13662.359,E2 -13662.359} C_VEL
LIN {X 0,Y 347.903,Z 214.462,A -85,B 0,C 180,E1 -13665.97,E2 -13665.97} C_VEL
LIN {X 0,Y 347.9,Z 214.459,A -85,B 0,C 180,E1 -13669.524,E2 -13669.524} C_VEL
LIN {X 0,Y 348.094,Z 214.439,A -85,B 0,C 180,E1 -13673.041,E2 -13673.041} C_VEL
LIN {X 0,Y 348.206,Z 214.425,A -85,B 0,C 180,E1 -13677.686,E2 -13677.686} C_VEL
LIN {X 0,Y 348.307,Z 214.411,A -85,B 0,C 180,E1 -13679.999,E2 -13679.999} C_VEL
LIN {X 0,Y 348.206,Z 214.421,A -85,B 0,C 180,E1 -13682.313,E2 -13682.313} C_VEL
LIN {X 0,Y 348.078,Z 214.436,A -85,B 0,C 180,E1 -13686.958,E2 -13686.958} C_VEL
LIN {X 0,Y 347.897,Z 214.456,A -85,B 0,C 180,E1 -13690.475,E2 -13690.475} C_VEL
LIN {X 0,Y 347.902,Z 214.462,A -85,B 0,C 180,E1 -13694.149,E2 -13694.149} C_VEL
LIN {X 0,Y 347.831,Z 214.468,A -85,B 0,C 180,E1 -13698.258,E2 -13698.258} C_VEL
LIN {X 0,Y 347.77,Z 214.473,A -85,B 0,C 180,E1 -13701.625,E2 -13701.625} C_VEL
LIN {X 0,Y 347.814,Z 214.469,A -85,B 0,C 180,E1 -13705.108,E2 -13705.108} C_VEL
LIN {X 0,Y 347.81,Z 214.471,A -85,B 0,C 180,E1 -13707.693,E2 -13707.693} C_VEL
LIN {X 0,Y 347.749,Z 214.479,A -85,B 0,C 180,E1 -13710.347,E2 -13710.347} C_VEL
LIN {X 0,Y 347.751,Z 214.476,A -85,B 0,C 180,E1 -13714.043,E2 -13714.043} C_VEL
LIN {X 0,Y 347.763,Z 214.481,A -85,B 0,C 180,E1 -13717.32,E2 -13717.32} C_VEL
LIN {X 0,Y 347.73,Z 214.476,A -85,B 0,C 180,E1 -13720.297,E2 -13720.297} C_VEL
LIN {X 0,Y 347.725,Z 214.485,A -85,B 0,C 180,E1 -13723.407,E2 -13723.407} C_VEL
LIN {X 0,Y 347.741,Z 214.579,A -85,B 0,C 180,E1 -13724.677,E2 -13724.677} C_VEL
LIN {X 0,Y 348.087,Z 216.036,A -85,B 0,C 180,E1 -13725.034,E2 -13725.034} C_VEL
LIN {X 0,Y 350.091,Z 220.54,A -85,B 0,C 180,E1 -13726.276,E2 -13726.276} C_VEL
LIN {X 0,Y 352.826,Z 227.268,A -85,B 0,C 180,E1 -13727.972,E2 -13727.972} C_VEL
LIN {X 0,Y 362.282,Z 242.699,A -85,B 0,C 180,E1 -13729.907,E2 -13729.907} C_VEL
LIN {X 0,Y 370.231,Z 257.36,A -85,B 0,C 180,E1 -13731.435,E2 -13731.435} C_VEL
LIN {X 0,Y 377.152,Z 271.564,A -85,B 0,C 180,E1 -13732.712,E2 -13732.712} C_VEL
LIN {X 0,Y 378.887,Z 275.577,A -85,B 0,C 180,E1 -13733.03,E2 -13733.03} C_VEL
LIN {X 0,Y 378.756,Z 283.107,A -85,B 0,C 180,E1 -13733.203,E2 -13733.203} C_VEL
LIN {X 0,Y 372.985,Z 436.42,A -85,B 0,C 180,E1 -13736.351,E2 -13736.351} C_VEL
LIN {X 0,Y 371.631,Z 452.533,A -85,B 0,C 180,E1 -13736.861,E2 -13736.861} C_VEL
LIN {X 0,Y 369.762,Z 469.231,A -85,B 0,C 180,E1 -13737.603,E2 -13737.603} C_VEL
LIN {X 0,Y 367.902,Z 483.889,A -85,B 0,C 180,E1 -13738.468,E2 -13738.468} C_VEL
LIN {X 0,Y 365.615,Z 498.609,A -85,B 0,C 180,E1 -13739.535,E2 -13739.535} C_VEL
LIN {X 0,Y 363.015,Z 513.681,A -85,B 0,C 180,E1 -13740.895,E2 -13740.895} C_VEL
LIN {X 0,Y 360.565,Z 526.324,A -85,B 0,C 180,E1 -13742.264,E2 -13742.264} C_VEL
LIN {X 0,Y 358.137,Z 538.394,A -85,B 0,C 180,E1 -13743.796,E2 -13743.796} C_VEL
LIN {X 0,Y 355.513,Z 551.474,A -85,B 0,C 180,E1 -13745.781,E2 -13745.781} C_VEL
LIN {X 0,Y 353.171,Z 562.52,A -85,B 0,C 180,E1 -13747.782,E2 -13747.782} C_VEL
LIN {X 0,Y 351.244,Z 572.01,A -85,B 0,C 180,E1 -13749.807,E2 -13749.807} C_VEL
LIN {X 0,Y 349.551,Z 581.269,A -85,B 0,C 180,E1 -13752.143,E2 -13752.143} C_VEL
LIN {X 0,Y 348.05,Z 589.89,A -85,B 0,C 180,E1 -13754.779,E2 -13754.779} C_VEL
LIN {X 0,Y 347.191,Z 596.12,A -85,B 0,C 180,E1 -13757.132,E2 -13757.132} C_VEL
LIN {X 0,Y 346.516,Z 601.188,A -85,B 0,C 180,E1 -13759.48,E2 -13759.48} C_VEL
LIN {X 0,Y 346.266,Z 605.175,A -85,B 0,C 180,E1 -13761.83,E2 -13761.83} C_VEL
LIN {X 0,Y 346.159,Z 608.068,A -85,B 0,C 180,E1 -13764.171,E2 -13764.171} C_VEL
LIN {X 0,Y 346.114,Z 610.002,A -85,B 0,C 180,E1 -13766.505,E2 -13766.505} C_VEL
LIN {X 0,Y 346.118,Z 610.89,A -85,B 0,C 180,E1 -13768.834,E2 -13768.834} C_VEL
LIN {X 0,Y 346.121,Z 610.859,A -85,B 0,C 180,E1 -13771.161,E2 -13771.161} C_VEL
LIN {X 0,Y 346.113,Z 609.781,A -85,B 0,C 180,E1 -13773.489,E2 -13773.489} C_VEL
LIN {X 0,Y 346.155,Z 607.772,A -85,B 0,C 180,E1 -13775.823,E2 -13775.823} C_VEL
LIN {X 0,Y 346.261,Z 604.662,A -85,B 0,C 180,E1 -13778.165,E2 -13778.165} C_VEL
LIN {X 0,Y 346.494,Z 600.556,A -85,B 0,C 180,E1 -13780.515,E2 -13780.515} C_VEL
LIN {X 0,Y 347.338,Z 593.945,A -85,B 0,C 180,E1 -13783.38,E2 -13783.38} C_VEL
LIN {X 0,Y 348.223,Z 586.858,A -85,B 0,C 180,E1 -13785.807,E2 -13785.807} C_VEL
LIN {X 0,Y 349.635,Z 578.583,A -85,B 0,C 180,E1 -13788.15,E2 -13788.15} C_VEL
LIN {X 0,Y 351.308,Z 568.704,A -85,B 0,C 180,E1 -13790.489,E2 -13790.489} C_VEL
LIN {X 0,Y 353.254,Z 558.542,A -85,B 0,C 180,E1 -13792.514,E2 -13792.514} C_VEL
LIN {X 0,Y 355.488,Z 546.518,A -85,B 0,C 180,E1 -13794.526,E2 -13794.526} C_VEL
LIN {X 0,Y 357.57,Z 535.521,A -85,B 0,C 180,E1 -13796.086,E2 -13796.086} C_VEL
LIN {X 0,Y 359.878,Z 522.85,A -85,B 0,C 180,E1 -13797.629,E2 -13797.629} C_VEL
LIN {X 0,Y 362.362,Z 508.334,A -85,B 0,C 180,E1 -13799.094,E2 -13799.094} C_VEL
LIN {X 0,Y 364.739,Z 492.697,A -85,B 0,C 180,E1 -13800.38,E2 -13800.38} C_VEL
LIN {X 0,Y 366.773,Z 477.333,A -85,B 0,C 180,E1 -13801.392,E2 -13801.392} C_VEL
LIN {X 0,Y 368.53,Z 461.1,A -85,B 0,C 180,E1 -13802.229,E2 -13802.229} C_VEL
LIN {X 0,Y 369.962,Z 445.639,A -85,B 0,C 180,E1 -13802.815,E2 -13802.815} C_VEL
LIN {X 0,Y 370.923,Z 429.011,A -85,B 0,C 180,E1 -13803.245,E2 -13803.245} C_VEL
LIN {X 0,Y 375.949,Z 275.406,A -85,B 0,C 180,E1 -13806.332,E2 -13806.332} C_VEL
LIN {X 0,Y 375.194,Z 272.513,A -85,B 0,C 180,E1 -13806.479,E2 -13806.479} C_VEL
LIN {X 0,Y 365.337,Z 252.052,A -85,B 0,C 180,E1 -13808.047,E2 -13808.047} C_VEL
LIN {X 0,Y 354.787,Z 232.291,A -85,B 0,C 180,E1 -13809.794,E2 -13809.794} C_VEL
LIN {X 0,Y 352.779,Z 228.526,A -85,B 0,C 180,E1 -13810.166,E2 -13810.166} C_VEL
LIN {X 0,Y 347.703,Z 214.479,A -85,B 0,C 180,E1 -13813.205,E2 -13813.205} C_VEL
LIN {X 0,Y 347.711,Z 214.481,A -85,B 0,C 180,E1 -13816.682,E2 -13816.682} C_VEL
LIN {X 0,Y 347.735,Z 214.476,A -85,B 0,C 180,E1 -13820.169,E2 -13820.169} C_VEL
LIN {X 0,Y 347.746,Z 214.467,A -85,B 0,C 180,E1 -13823.933,E2 -13823.933} C_VEL
LIN {X 0,Y 347.707,Z 214.474,A -85,B 0,C 180,E1 -13826.926,E2 -13826.926} C_VEL
LIN {X 0,Y 347.751,Z 214.484,A -85,B 0,C 180,E1 -13830.986,E2 -13830.986} C_VEL
LIN {X 0,Y 347.803,Z 214.451,A -85,B 0,C 180,E1 -13833.606,E2 -13833.606} C_VEL
LIN {X 0,Y 347.771,Z 214.477,A -85,B 0,C 180,E1 -13836.161,E2 -13836.161} C_VEL
LIN {X 0,Y 347.807,Z 214.445,A -85,B 0,C 180,E1 -13839.91,E2 -13839.91} C_VEL
LIN {X 0,Y 347.837,Z 214.461,A -85,B 0,C 180,E1 -13842.358,E2 -13842.358} C_VEL
LIN {X 0,Y 347.868,Z 214.449,A -85,B 0,C 180,E1 -13845.97,E2 -13845.97} C_VEL
LIN {X 0,Y 347.903,Z 214.443,A -85,B 0,C 180,E1 -13849.525,E2 -13849.525} C_VEL
LIN {X 0,Y 348.067,Z 214.436,A -85,B 0,C 180,E1 -13853.042,E2 -13853.042} C_VEL
LIN {X 0,Y 348.177,Z 214.398,A -85,B 0,C 180,E1 -13857.687,E2 -13857.687} C_VEL
LIN {X 0,Y 348.316,Z 214.405,A -85,B 0,C 180,E1 -13860.001,E2 -13860.001} C_VEL
LIN {X 0,Y 348.177,Z 214.423,A -85,B 0,C 180,E1 -13862.314,E2 -13862.314} C_VEL
LIN {X 0,Y 348.062,Z 214.439,A -85,B 0,C 180,E1 -13866.959,E2 -13866.959} C_VEL
LIN {X 0,Y 347.899,Z 214.443,A -85,B 0,C 180,E1 -13870.476,E2 -13870.476} C_VEL
LIN {X 0,Y 347.871,Z 214.458,A -85,B 0,C 180,E1 -13874.152,E2 -13874.152} C_VEL
LIN {X 0,Y 347.864,Z 214.444,A -85,B 0,C 180,E1 -13878.292,E2 -13878.292} C_VEL
LIN {X 0,Y 347.762,Z 214.474,A -85,B 0,C 180,E1 -13881.637,E2 -13881.637} C_VEL
LIN {X 0,Y 347.787,Z 214.457,A -85,B 0,C 180,E1 -13885.111,E2 -13885.111} C_VEL
LIN {X 0,Y 347.786,Z 214.466,A -85,B 0,C 180,E1 -13887.697,E2 -13887.697} C_VEL
LIN {X 0,Y 347.741,Z 214.48,A -85,B 0,C 180,E1 -13890.349,E2 -13890.349} C_VEL
LIN {X 0,Y 347.723,Z 214.474,A -85,B 0,C 180,E1 -13894.467,E2 -13894.467} C_VEL
LIN {X 0,Y 347.752,Z 214.469,A -85,B 0,C 180,E1 -13897.992,E2 -13897.992} C_VEL
LIN {X 0,Y 347.733,Z 214.481,A -85,B 0,C 180,E1 -13901.834,E2 -13901.834} C_VEL
LIN {X 0,Y 347.688,Z 214.469,A -85,B 0,C 180,E1 -13905.031,E2 -13905.031} C_VEL
LIN {X 0,Y 347.733,Z 214.482,A -85,B 0,C 180,E1 -13908.401,E2 -13908.401} C_VEL
LIN {X 0,Y 347.752,Z 214.474,A -85,B 0,C 180,E1 -13912.017,E2 -13912.017} C_VEL
LIN {X 0,Y 347.734,Z 214.468,A -85,B 0,C 180,E1 -13915.54,E2 -13915.54} C_VEL
LIN {X 0,Y 347.736,Z 214.482,A -85,B 0,C 180,E1 -13918.304,E2 -13918.304} C_VEL
LIN {X 0,Y 347.739,Z 214.476,A -85,B 0,C 180,E1 -13920.988,E2 -13920.988} C_VEL
LIN {X 0,Y 347.744,Z 214.474,A -85,B 0,C 180,E1 -13923.605,E2 -13923.605} C_VEL
LIN {X 0,Y 347.761,Z 214.479,A -85,B 0,C 180,E1 -13926.164,E2 -13926.164} C_VEL
LIN {X 0,Y 347.795,Z 214.473,A -85,B 0,C 180,E1 -13929.912,E2 -13929.912} C_VEL
LIN {X 0,Y 347.831,Z 214.473,A -85,B 0,C 180,E1 -13932.361,E2 -13932.361} C_VEL
LIN {X 0,Y 347.894,Z 214.458,A -85,B 0,C 180,E1 -13936.332,E2 -13936.332} C_VEL
LIN {X 0,Y 348.999,Z 217.467,A -85,B 0,C 180,E1 -13936.582,E2 -13936.582} C_VEL
LIN {X 0,Y 350.517,Z 219.48,A -85,B 0,C 180,E1 -13936.832,E2 -13936.832} C_VEL
LIN {X 0,Y 362.257,Z 238.622,A -85,B 0,C 180,E1 -13938.758,E2 -13938.758} C_VEL
LIN {X 0,Y 370.497,Z 254.49,A -85,B 0,C 180,E1 -13940.082,E2 -13940.082} C_VEL
LIN {X 0,Y 376.046,Z 266.245,A -85,B 0,C 180,E1 -13940.955,E2 -13940.955} C_VEL
LIN {X 0,Y 370.871,Z 418.257,A -85,B 0,C 180,E1 -13944.02,E2 -13944.02} C_VEL
LIN {X 0,Y 369.734,Z 435.369,A -85,B 0,C 180,E1 -13944.583,E2 -13944.583} C_VEL
LIN {X 0,Y 368.305,Z 450.619,A -85,B 0,C 180,E1 -13945.283,E2 -13945.283} C_VEL
LIN {X 0,Y 366.398,Z 467.512,A -85,B 0,C 180,E1 -13946.301,E2 -13946.301} C_VEL
LIN {X 0,Y 364.245,Z 483.36,A -85,B 0,C 180,E1 -13947.515,E2 -13947.515} C_VEL
LIN {X 0,Y 361.938,Z 498.011,A -85,B 0,C 180,E1 -13948.89,E2 -13948.89} C_VEL
LIN {X 0,Y 359.632,Z 511.325,A -85,B 0,C 180,E1 -13950.396,E2 -13950.396} C_VEL
LIN {X 0,Y 357.418,Z 523.04,A -85,B 0,C 180,E1 -13951.974,E2 -13951.974} C_VEL
LIN {X 0,Y 355.045,Z 535.591,A -85,B 0,C 180,E1 -13953.975,E2 -13953.975} C_VEL
LIN {X 0,Y 352.993,Z 546.169,A -85,B 0,C 180,E1 -13955.973,E2 -13955.973} C_VEL
LIN {X 0,Y 350.97,Z 556.691,A -85,B 0,C 180,E1 -13958.35,E2 -13958.35} C_VEL
LIN {X 0,Y 349.414,Z 565.372,A -85,B 0,C 180,E1 -13960.725,E2 -13960.725} C_VEL
LIN {X 0,Y 348.331,Z 571.75,A -85,B 0,C 180,E1 -13962.825,E2 -13962.825} C_VEL
LIN {X 0,Y 347.703,Z 575.711,A -85,B 0,C 180,E1 -13964.337,E2 -13964.337} C_VEL
LIN {X 0,Y 346.671,Z 577.915,A -85,B 0,C 180,E1 -13965.229,E2 -13965.229} C_VEL
LIN {X 0,Y 343.367,Z 581.181,A -85,B 0,C 180,E1 -13966.685,E2 -13966.685} C_VEL
LIN {X 0,Y 340.698,Z 583.506,A -85,B 0,C 180,E1 -13967.88,E2 -13967.88} C_VEL
LIN {X 0,Y 339.504,Z 585.005,A -85,B 0,C 180,E1 -13968.822,E2 -13968.822} C_VEL
LIN {X 0,Y 339.372,Z 585.488,A -85,B 0,C 180,E1 -13969.144,E2 -13969.144} C_VEL
LIN {X 0,Y 338.914,Z 588.719,A -85,B 0,C 180,E1 -13971.919,E2 -13971.919} C_VEL
LIN {X 0,Y 338.723,Z 590.557,A -85,B 0,C 180,E1 -13974.52,E2 -13974.52} C_VEL
LIN {X 0,Y 338.754,Z 591.259,A -85,B 0,C 180,E1 -13977.159,E2 -13977.159} C_VEL
LIN {X 0,Y 338.825,Z 590.71,A -85,B 0,C 180,E1 -13979.857,E2 -13979.857} C_VEL
LIN {X 0,Y 339.027,Z 588.917,A -85,B 0,C 180,E1 -13982.616,E2 -13982.616} C_VEL
LIN {X 0,Y 339.482,Z 585.756,A -85,B 0,C 180,E1 -13985.429,E2 -13985.429} C_VEL
LIN {X 0,Y 340.038,Z 582.371,A -85,B 0,C 180,E1 -13987.564,E2 -13987.564} C_VEL
LIN {X 0,Y 341.008,Z 576.786,A -85,B 0,C 180,E1 -13990.309,E2 -13990.309} C_VEL
LIN {X 0,Y 342.135,Z 570.765,A -85,B 0,C 180,E1 -13992.679,E2 -13992.679} C_VEL
LIN {X 0,Y 343.817,Z 562.621,A -85,B 0,C 180,E1 -13995.263,E2 -13995.263} C_VEL
LIN {X 0,Y 345.757,Z 553.989,A -85,B 0,C 180,E1 -13997.519,E2 -13997.519} C_VEL
LIN {X 0,Y 348,Z 543.92,A -85,B 0,C 180,E1 -13999.74,E2 -13999.74} C_VEL
LIN {X 0,Y 350.639,Z 532.325,A -85,B 0,C 180,E1 -14001.879,E2 -14001.879} C_VEL
LIN {X 0,Y 353.372,Z 520.027,A -85,B 0,C 180,E1 -14003.777,E2 -14003.777} C_VEL
LIN {X 0,Y 356.068,Z 506.833,A -85,B 0,C 180,E1 -14005.474,E2 -14005.474} C_VEL
LIN {X 0,Y 358.709,Z 492.947,A -85,B 0,C 180,E1 -14006.96,E2 -14006.96} C_VEL
LIN {X 0,Y 361.25,Z 477.649,A -85,B 0,C 180,E1 -14008.312,E2 -14008.312} C_VEL
LIN {X 0,Y 363.48,Z 462.808,A -85,B 0,C 180,E1 -14009.365,E2 -14009.365} C_VEL
LIN {X 0,Y 365.326,Z 447.442,A -85,B 0,C 180,E1 -14010.24,E2 -14010.24} C_VEL
LIN {X 0,Y 366.844,Z 430.976,A -85,B 0,C 180,E1 -14010.938,E2 -14010.938} C_VEL
LIN {X 0,Y 367.93,Z 414.834,A -85,B 0,C 180,E1 -14011.408,E2 -14011.408} C_VEL
LIN {X 0,Y 373.573,Z 270.217,A -85,B 0,C 180,E1 -14014.416,E2 -14014.416} C_VEL
LIN {X 0,Y 365.999,Z 255.204,A -85,B 0,C 180,E1 -14015.847,E2 -14015.847} C_VEL
LIN {X 0,Y 358.089,Z 241.43,A -85,B 0,C 180,E1 -14017.402,E2 -14017.402} C_VEL
LIN {X 0,Y 352.646,Z 233.051,A -85,B 0,C 180,E1 -14018.518,E2 -14018.518} C_VEL
LIN {X 0,Y 349.143,Z 228.147,A -85,B 0,C 180,E1 -14019.258,E2 -14019.258} C_VEL
LIN {X 0,Y 346.673,Z 224.567,A -85,B 0,C 180,E1 -14019.801,E2 -14019.801} C_VEL
LIN {X 0,Y 344.449,Z 221.467,A -85,B 0,C 180,E1 -14020.303,E2 -14020.303} C_VEL
LIN {X 0,Y 343.633,Z 220.212,A -85,B 0,C 180,E1 -14020.493,E2 -14020.493} C_VEL
LIN {X 0,Y 341.67,Z 217.959,A -85,B 0,C 180,E1 -14020.933,E2 -14020.933} C_VEL
LIN {X 0,Y 340.833,Z 215.34,A -85,B 0,C 180,E1 -14021.213,E2 -14021.213} C_VEL
LIN {X 0,Y 340.868,Z 215.336,A -85,B 0,C 180,E1 -14025.675,E2 -14025.675} C_VEL
LIN {X 0,Y 340.852,Z 215.337,A -85,B 0,C 180,E1 -14029.305,E2 -14029.305} C_VEL
LIN {X 0,Y 341.062,Z 215.314,A -85,B 0,C 180,E1 -14032.897,E2 -14032.897} C_VEL
LIN {X 0,Y 341.168,Z 215.302,A -85,B 0,C 180,E1 -14037.638,E2 -14037.638} C_VEL
LIN {X 0,Y 341.259,Z 215.289,A -85,B 0,C 180,E1 -14039.999,E2 -14039.999} C_VEL
LIN {X 0,Y 341.168,Z 215.298,A -85,B 0,C 180,E1 -14042.361,E2 -14042.361} C_VEL
LIN {X 0,Y 341.025,Z 215.313,A -85,B 0,C 180,E1 -14047.102,E2 -14047.102} C_VEL
LIN {X 0,Y 340.849,Z 215.334,A -85,B 0,C 180,E1 -14050.694,E2 -14050.694} C_VEL
LIN {X 0,Y 340.867,Z 215.338,A -85,B 0,C 180,E1 -14054.324,E2 -14054.324} C_VEL
LIN {X 0,Y 340.788,Z 215.344,A -85,B 0,C 180,E1 -14058.439,E2 -14058.439} C_VEL
LIN {X 0,Y 340.721,Z 215.35,A -85,B 0,C 180,E1 -14061.841,E2 -14061.841} C_VEL
LIN {X 0,Y 340.774,Z 215.351,A -85,B 0,C 180,E1 -14065.664,E2 -14065.664} C_VEL
LIN {X 0,Y 340.73,Z 215.355,A -85,B 0,C 180,E1 -14068.32,E2 -14068.32} C_VEL
LIN {X 0,Y 340.699,Z 215.36,A -85,B 0,C 180,E1 -14071.044,E2 -14071.044} C_VEL
LIN {X 0,Y 340.72,Z 215.358,A -85,B 0,C 180,E1 -14075.278,E2 -14075.278} C_VEL
LIN {X 0,Y 340.711,Z 215.355,A -85,B 0,C 180,E1 -14078.385,E2 -14078.385} C_VEL
LIN {X 0,Y 340.699,Z 215.349,A -85,B 0,C 180,E1 -14082.044,E2 -14082.044} C_VEL
LIN {X 0,Y 340.695,Z 215.435,A -85,B 0,C 180,E1 -14083.495,E2 -14083.495} C_VEL
LIN {X 0,Y 345.362,Z 226.949,A -85,B 0,C 180,E1 -14086.676,E2 -14086.676} C_VEL
LIN {X 0,Y 352.757,Z 238.646,A -85,B 0,C 180,E1 -14088.306,E2 -14088.306} C_VEL
LIN {X 0,Y 358.885,Z 249.068,A -85,B 0,C 180,E1 -14089.577,E2 -14089.577} C_VEL
LIN {X 0,Y 365.965,Z 262.31,A -85,B 0,C 180,E1 -14090.979,E2 -14090.979} C_VEL
LIN {X 0,Y 372.972,Z 276.957,A -85,B 0,C 180,E1 -14092.317,E2 -14092.317} C_VEL
LIN {X 0,Y 373.451,Z 277.982,A -85,B 0,C 180,E1 -14092.406,E2 -14092.406} C_VEL
LIN {X 0,Y 367.242,Z 436.013,A -85,B 0,C 180,E1 -14095.698,E2 -14095.698} C_VEL
LIN {X 0,Y 365.844,Z 452.398,A -85,B 0,C 180,E1 -14096.226,E2 -14096.226} C_VEL
LIN {X 0,Y 363.966,Z 468.394,A -85,B 0,C 180,E1 -14096.94,E2 -14096.94} C_VEL
LIN {X 0,Y 361.873,Z 484.181,A -85,B 0,C 180,E1 -14097.881,E2 -14097.881} C_VEL
LIN {X 0,Y 359.507,Z 498.808,A -85,B 0,C 180,E1 -14098.96,E2 -14098.96} C_VEL
LIN {X 0,Y 356.923,Z 513.052,A -85,B 0,C 180,E1 -14100.26,E2 -14100.26} C_VEL
LIN {X 0,Y 354.261,Z 526.412,A -85,B 0,C 180,E1 -14101.727,E2 -14101.727} C_VEL
LIN {X 0,Y 351.758,Z 538.423,A -85,B 0,C 180,E1 -14103.284,E2 -14103.284} C_VEL
LIN {X 0,Y 349.317,Z 549.679,A -85,B 0,C 180,E1 -14105.005,E2 -14105.005} C_VEL
LIN {X 0,Y 346.854,Z 560.964,A -85,B 0,C 180,E1 -14107.041,E2 -14107.041} C_VEL
LIN {X 0,Y 344.47,Z 571.927,A -85,B 0,C 180,E1 -14109.392,E2 -14109.392} C_VEL
LIN {X 0,Y 342.716,Z 581.165,A -85,B 0,C 180,E1 -14111.774,E2 -14111.774} C_VEL
LIN {X 0,Y 341.105,Z 589.765,A -85,B 0,C 180,E1 -14114.461,E2 -14114.461} C_VEL
LIN {X 0,Y 340.201,Z 595.978,A -85,B 0,C 180,E1 -14116.863,E2 -14116.863} C_VEL
LIN {X 0,Y 339.467,Z 601.026,A -85,B 0,C 180,E1 -14119.259,E2 -14119.259} C_VEL
LIN {X 0,Y 339.19,Z 605.007,A -85,B 0,C 180,E1 -14121.658,E2 -14121.658} C_VEL
LIN {X 0,Y 339.061,Z 608.059,A -85,B 0,C 180,E1 -14124.226,E2 -14124.226} C_VEL
LIN {X 0,Y 339.037,Z 609.815,A -85,B 0,C 180,E1 -14126.432,E2 -14126.432} C_VEL
LIN {X 0,Y 339.02,Z 610.688,A -85,B 0,C 180,E1 -14128.809,E2 -14128.809} C_VEL
LIN {X 0,Y 339.023,Z 610.649,A -85,B 0,C 180,E1 -14131.185,E2 -14131.185} C_VEL
LIN {X 0,Y 339.036,Z 609.556,A -85,B 0,C 180,E1 -14133.562,E2 -14133.562} C_VEL
LIN {X 0,Y 339.081,Z 607.538,A -85,B 0,C 180,E1 -14135.945,E2 -14135.945} C_VEL
LIN {X 0,Y 339.186,Z 604.408,A -85,B 0,C 180,E1 -14138.336,E2 -14138.336} C_VEL
LIN {X 0,Y 339.443,Z 600.284,A -85,B 0,C 180,E1 -14140.736,E2 -14140.736} C_VEL
LIN {X 0,Y 340.164,Z 594.937,A -85,B 0,C 180,E1 -14143.133,E2 -14143.133} C_VEL
LIN {X 0,Y 341.002,Z 588.387,A -85,B 0,C 180,E1 -14145.537,E2 -14145.537} C_VEL
LIN {X 0,Y 342.412,Z 580.514,A -85,B 0,C 180,E1 -14147.927,E2 -14147.927} C_VEL
LIN {X 0,Y 344.051,Z 571.003,A -85,B 0,C 180,E1 -14150.316,E2 -14150.316} C_VEL
LIN {X 0,Y 345.98,Z 561.177,A -85,B 0,C 180,E1 -14152.384,E2 -14152.384} C_VEL
LIN {X 0,Y 348.41,Z 548.871,A -85,B 0,C 180,E1 -14154.566,E2 -14154.566} C_VEL
LIN {X 0,Y 350.69,Z 537.182,A -85,B 0,C 180,E1 -14156.317,E2 -14156.317} C_VEL
LIN {X 0,Y 353.291,Z 523.542,A -85,B 0,C 180,E1 -14158.028,E2 -14158.028} C_VEL
LIN {X 0,Y 355.93,Z 508.551,A -85,B 0,C 180,E1 -14159.575,E2 -14159.575} C_VEL
LIN {X 0,Y 358.278,Z 493.738,A -85,B 0,C 180,E1 -14160.824,E2 -14160.824} C_VEL
LIN {X 0,Y 360.511,Z 477.581,A -85,B 0,C 180,E1 -14161.919,E2 -14161.919} C_VEL
LIN {X 0,Y 362.402,Z 460.743,A -85,B 0,C 180,E1 -14162.801,E2 -14162.801} C_VEL
LIN {X 0,Y 363.882,Z 445.216,A -85,B 0,C 180,E1 -14163.393,E2 -14163.393} C_VEL
LIN {X 0,Y 364.865,Z 428.531,A -85,B 0,C 180,E1 -14163.829,E2 -14163.829} C_VEL
LIN {X 0,Y 370.058,Z 277.343,A -85,B 0,C 180,E1 -14166.906,E2 -14166.906} C_VEL
LIN {X 0,Y 369.6,Z 275.484,A -85,B 0,C 180,E1 -14167.001,E2 -14167.001} C_VEL
LIN {X 0,Y 360.405,Z 256.262,A -85,B 0,C 180,E1 -14168.507,E2 -14168.507} C_VEL
LIN {X 0,Y 350.018,Z 236.688,A -85,B 0,C 180,E1 -14170.271,E2 -14170.271} C_VEL
LIN {X 0,Y 345.303,Z 228.218,A -85,B 0,C 180,E1 -14171.144,E2 -14171.144} C_VEL
LIN {X 0,Y 341.378,Z 217.693,A -85,B 0,C 180,E1 -14173.489,E2 -14173.489} C_VEL
LIN {X 0,Y 340.624,Z 215.37,A -85,B 0,C 180,E1 -14174.049,E2 -14174.049} C_VEL
LIN {X 0,Y 340.707,Z 215.357,A -85,B 0,C 180,E1 -14177.946,E2 -14177.946} C_VEL
LIN {X 0,Y 340.715,Z 215.356,A -85,B 0,C 180,E1 -14181.771,E2 -14181.771} C_VEL
LIN {X 0,Y 340.698,Z 215.36,A -85,B 0,C 180,E1 -14185.593,E2 -14185.593} C_VEL
LIN {X 0,Y 340.67,Z 215.346,A -85,B 0,C 180,E1 -14188.953,E2 -14188.953} C_VEL
LIN {X 0,Y 340.776,Z 215.329,A -85,B 0,C 180,E1 -14193.018,E2 -14193.018} C_VEL
LIN {X 0,Y 340.752,Z 215.349,A -85,B 0,C 180,E1 -14195.639,E2 -14195.639} C_VEL
LIN {X 0,Y 340.749,Z 215.327,A -85,B 0,C 180,E1 -14199.475,E2 -14199.475} C_VEL
LIN {X 0,Y 340.829,Z 215.332,A -85,B 0,C 180,E1 -14201.983,E2 -14201.983} C_VEL
LIN {X 0,Y 340.84,Z 215.33,A -85,B 0,C 180,E1 -14205.704,E2 -14205.704} C_VEL
LIN {X 0,Y 340.845,Z 215.316,A -85,B 0,C 180,E1 -14209.306,E2 -14209.306} C_VEL
LIN {X 0,Y 341.034,Z 215.313,A -85,B 0,C 180,E1 -14212.898,E2 -14212.898} C_VEL
LIN {X 0,Y 341.139,Z 215.273,A -85,B 0,C 180,E1 -14217.639,E2 -14217.639} C_VEL
LIN {X 0,Y 341.267,Z 215.284,A -85,B 0,C 180,E1 -14220.001,E2 -14220.001} C_VEL
LIN {X 0,Y 341.139,Z 215.299,A -85,B 0,C 180,E1 -14222.362,E2 -14222.362} C_VEL
LIN {X 0,Y 341.03,Z 215.316,A -85,B 0,C 180,E1 -14227.103,E2 -14227.103} C_VEL
LIN {X 0,Y 340.841,Z 215.319,A -85,B 0,C 180,E1 -14230.695,E2 -14230.695} C_VEL
LIN {X 0,Y 340.836,Z 215.336,A -85,B 0,C 180,E1 -14234.327,E2 -14234.327} C_VEL
LIN {X 0,Y 340.81,Z 215.321,A -85,B 0,C 180,E1 -14238.468,E2 -14238.468} C_VEL
LIN {X 0,Y 340.729,Z 215.351,A -85,B 0,C 180,E1 -14241.859,E2 -14241.859} C_VEL
LIN {X 0,Y 340.747,Z 215.33,A -85,B 0,C 180,E1 -14245.667,E2 -14245.667} C_VEL
LIN {X 0,Y 340.717,Z 215.351,A -85,B 0,C 180,E1 -14248.323,E2 -14248.323} C_VEL
LIN {X 0,Y 340.681,Z 215.353,A -85,B 0,C 180,E1 -14251.047,E2 -14251.047} C_VEL
LIN {X 0,Y 340.697,Z 215.356,A -85,B 0,C 180,E1 -14255.282,E2 -14255.282} C_VEL
LIN {X 0,Y 340.689,Z 215.342,A -85,B 0,C 180,E1 -14258.389,E2 -14258.389} C_VEL
LIN {X 0,Y 340.681,Z 215.361,A -85,B 0,C 180,E1 -14262.049,E2 -14262.049} C_VEL
LIN {X 0,Y 340.636,Z 215.354,A -85,B 0,C 180,E1 -14266.231,E2 -14266.231} C_VEL
LIN {X 0,Y 340.661,Z 215.353,A -85,B 0,C 180,E1 -14269.76,E2 -14269.76} C_VEL
LIN {X 0,Y 340.692,Z 215.359,A -85,B 0,C 180,E1 -14273.262,E2 -14273.262} C_VEL
LIN {X 0,Y 340.682,Z 215.348,A -85,B 0,C 180,E1 -14276.157,E2 -14276.157} C_VEL
LIN {X 0,Y 340.715,Z 215.346,A -85,B 0,C 180,E1 -14280.038,E2 -14280.038} C_VEL
LIN {X 0,Y 340.714,Z 215.355,A -85,B 0,C 180,E1 -14283.017,E2 -14283.017} C_VEL
LIN {X 0,Y 340.735,Z 215.354,A -85,B 0,C 180,E1 -14285.641,E2 -14285.641} C_VEL
LIN {X 0,Y 340.726,Z 215.358,A -85,B 0,C 180,E1 -14289.477,E2 -14289.477} C_VEL
LIN {X 0,Y 340.787,Z 215.35,A -85,B 0,C 180,E1 -14291.984,E2 -14291.984} C_VEL
LIN {X 0,Y 340.833,Z 215.341,A -85,B 0,C 180,E1 -14295.426,E2 -14295.426} C_VEL
LIN {X 0,Y 341.921,Z 218.313,A -85,B 0,C 180,E1 -14295.669,E2 -14295.669} C_VEL
LIN {X 0,Y 343.596,Z 220.52,A -85,B 0,C 180,E1 -14295.954,E2 -14295.954} C_VEL
LIN {X 0,Y 356.852,Z 241.922,A -85,B 0,C 180,E1 -14298.206,E2 -14298.206} C_VEL
LIN {X 0,Y 365.29,Z 258.139,A -85,B 0,C 180,E1 -14299.593,E2 -14299.593} C_VEL
LIN {X 0,Y 370.12,Z 268.373,A -85,B 0,C 180,E1 -14300.377,E2 -14300.377} C_VEL
LIN {X 0,Y 364.843,Z 417.898,A -85,B 0,C 180,E1 -14303.435,E2 -14303.435} C_VEL
LIN {X 0,Y 363.69,Z 434.384,A -85,B 0,C 180,E1 -14303.971,E2 -14303.971} C_VEL
LIN {X 0,Y 362.183,Z 450.564,A -85,B 0,C 180,E1 -14304.714,E2 -14304.714} C_VEL
LIN {X 0,Y 360.34,Z 466.377,A -85,B 0,C 180,E1 -14305.666,E2 -14305.666} C_VEL
LIN {X 0,Y 358.382,Z 481.008,A -85,B 0,C 180,E1 -14306.771,E2 -14306.771} C_VEL
LIN {X 0,Y 355.902,Z 496.102,A -85,B 0,C 180,E1 -14308.164,E2 -14308.164} C_VEL
LIN {X 0,Y 353.483,Z 509.867,A -85,B 0,C 180,E1 -14309.718,E2 -14309.718} C_VEL
LIN {X 0,Y 350.979,Z 522.68,A -85,B 0,C 180,E1 -14311.437,E2 -14311.437} C_VEL
LIN {X 0,Y 348.855,Z 533.682,A -85,B 0,C 180,E1 -14313.179,E2 -14313.179} C_VEL
LIN {X 0,Y 346.672,Z 544.316,A -85,B 0,C 180,E1 -14315.16,E2 -14315.16} C_VEL
LIN {X 0,Y 344.674,Z 554.11,A -85,B 0,C 180,E1 -14317.324,E2 -14317.324} C_VEL
LIN {X 0,Y 343.075,Z 562.225,A -85,B 0,C 180,E1 -14319.435,E2 -14319.435} C_VEL
LIN {X 0,Y 341.669,Z 570.048,A -85,B 0,C 180,E1 -14321.873,E2 -14321.873} C_VEL
LIN {X 0,Y 340.603,Z 576.469,A -85,B 0,C 180,E1 -14324.338,E2 -14324.338} C_VEL
LIN {X 0,Y 339.849,Z 581.703,A -85,B 0,C 180,E1 -14326.831,E2 -14326.831} C_VEL
LIN {X 0,Y 339.372,Z 585.488,A -85,B 0,C 180,E1 -14329.144,E2 -14329.144} C_VEL
LIN {X 0,Y 338.551,Z 586.847,A -85,B 0,C 180,E1 -14330.104,E2 -14330.104} C_VEL
LIN {X 0,Y 335.425,Z 588.67,A -85,B 0,C 180,E1 -14331.674,E2 -14331.674} C_VEL
LIN {X 0,Y 332.836,Z 589.801,A -85,B 0,C 180,E1 -14332.957,E2 -14332.957} C_VEL
LIN {X 0,Y 331.73,Z 590.505,A -85,B 0,C 180,E1 -14333.958,E2 -14333.958} C_VEL
LIN {X 0,Y 331.64,Z 590.678,A -85,B 0,C 180,E1 -14334.299,E2 -14334.299} C_VEL
LIN {X 0,Y 331.658,Z 591.456,A -85,B 0,C 180,E1 -14337.125,E2 -14337.125} C_VEL
LIN {X 0,Y 331.723,Z 591.013,A -85,B 0,C 180,E1 -14339.698,E2 -14339.698} C_VEL
LIN {X 0,Y 331.89,Z 589.703,A -85,B 0,C 180,E1 -14342.109,E2 -14342.109} C_VEL
LIN {X 0,Y 332.285,Z 586.994,A -85,B 0,C 180,E1 -14344.826,E2 -14344.826} C_VEL
LIN {X 0,Y 333.016,Z 582.732,A -85,B 0,C 180,E1 -14347.738,E2 -14347.738} C_VEL
LIN {X 0,Y 333.792,Z 578.51,A -85,B 0,C 180,E1 -14349.956,E2 -14349.956} C_VEL
LIN {X 0,Y 335.127,Z 571.681,A -85,B 0,C 180,E1 -14352.777,E2 -14352.777} C_VEL
LIN {X 0,Y 336.696,Z 564.367,A -85,B 0,C 180,E1 -14355.212,E2 -14355.212} C_VEL
LIN {X 0,Y 338.629,Z 556.306,A -85,B 0,C 180,E1 -14357.459,E2 -14357.459} C_VEL
LIN {X 0,Y 340.902,Z 546.686,A -85,B 0,C 180,E1 -14359.712,E2 -14359.712} C_VEL
LIN {X 0,Y 343.088,Z 537.388,A -85,B 0,C 180,E1 -14361.552,E2 -14361.552} C_VEL
LIN {X 0,Y 345.685,Z 526.377,A -85,B 0,C 180,E1 -14363.425,E2 -14363.425} C_VEL
LIN {X 0,Y 348.527,Z 513.552,A -85,B 0,C 180,E1 -14365.259,E2 -14365.259} C_VEL
LIN {X 0,Y 351.34,Z 499.986,A -85,B 0,C 180,E1 -14366.867,E2 -14366.867} C_VEL
LIN {X 0,Y 353.862,Z 486.665,A -85,B 0,C 180,E1 -14368.189,E2 -14368.189} C_VEL
LIN {X 0,Y 356.347,Z 471.673,A -85,B 0,C 180,E1 -14369.42,E2 -14369.42} C_VEL
LIN {X 0,Y 358.614,Z 455.769,A -85,B 0,C 180,E1 -14370.459,E2 -14370.459} C_VEL
LIN {X 0,Y 360.4,Z 439.619,A -85,B 0,C 180,E1 -14371.268,E2 -14371.268} C_VEL
LIN {X 0,Y 361.729,Z 423.668,A -85,B 0,C 180,E1 -14371.847,E2 -14371.847} C_VEL
LIN {X 0,Y 362.808,Z 401.74,A -85,B 0,C 180,E1 -14372.372,E2 -14372.372} C_VEL
LIN {X 0,Y 368.15,Z 272.88,A -85,B 0,C 180,E1 -14375.07,E2 -14375.07} C_VEL
LIN {X 0,Y 359.954,Z 256.631,A -85,B 0,C 180,E1 -14376.681,E2 -14376.681} C_VEL
LIN {X 0,Y 351.618,Z 242.39,A -85,B 0,C 180,E1 -14378.404,E2 -14378.404} C_VEL
LIN {X 0,Y 345.028,Z 232.916,A -85,B 0,C 180,E1 -14379.828,E2 -14379.828} C_VEL
LIN {X 0,Y 342.997,Z 229.942,A -85,B 0,C 180,E1 -14380.292,E2 -14380.292} C_VEL
LIN {X 0,Y 339.907,Z 225.648,A -85,B 0,C 180,E1 -14381.011,E2 -14381.011} C_VEL
LIN {X 0,Y 337.579,Z 222.396,A -85,B 0,C 180,E1 -14381.575,E2 -14381.575} C_VEL
LIN {X 0,Y 337.142,Z 221.357,A -85,B 0,C 180,E1 -14381.698,E2 -14381.698} C_VEL
LIN {X 0,Y 334.834,Z 219.123,A -85,B 0,C 180,E1 -14382.241,E2 -14382.241} C_VEL
LIN {X 0,Y 333.914,Z 216.947,A -85,B 0,C 180,E1 -14382.507,E2 -14382.507} C_VEL
LIN {X 0,Y 333.783,Z 216.206,A -85,B 0,C 180,E1 -14382.618,E2 -14382.618} C_VEL
LIN {X 0,Y 333.797,Z 216.218,A -85,B 0,C 180,E1 -14386.608,E2 -14386.608} C_VEL
LIN {X 0,Y 333.827,Z 216.217,A -85,B 0,C 180,E1 -14390.303,E2 -14390.303} C_VEL
LIN {X 0,Y 334.009,Z 216.193,A -85,B 0,C 180,E1 -14392.747,E2 -14392.747} C_VEL
LIN {X 0,Y 333.807,Z 216.218,A -85,B 0,C 180,E1 -14395.168,E2 -14395.168} C_VEL
LIN {X 0,Y 334.105,Z 216.181,A -85,B 0,C 180,E1 -14397.588,E2 -14397.588} C_VEL
LIN {X 0,Y 334.211,Z 216.167,A -85,B 0,C 180,E1 -14399.999,E2 -14399.999} C_VEL
LIN {X 0,Y 334.105,Z 216.178,A -85,B 0,C 180,E1 -14402.411,E2 -14402.411} C_VEL
LIN {X 0,Y 334.006,Z 216.193,A -85,B 0,C 180,E1 -14406.039,E2 -14406.039} C_VEL
LIN {X 0,Y 333.823,Z 216.211,A -85,B 0,C 180,E1 -14409.696,E2 -14409.696} C_VEL
LIN {X 0,Y 333.795,Z 216.213,A -85,B 0,C 180,E1 -14413.391,E2 -14413.391} C_VEL
LIN {X 0,Y 333.721,Z 216.227,A -85,B 0,C 180,E1 -14417.147,E2 -14417.147} C_VEL
LIN {X 0,Y 333.673,Z 216.232,A -85,B 0,C 180,E1 -14419.694,E2 -14419.694} C_VEL
LIN {X 0,Y 333.673,Z 216.231,A -85,B 0,C 180,E1 -14423.589,E2 -14423.589} C_VEL
LIN {X 0,Y 333.737,Z 216.225,A -85,B 0,C 180,E1 -14426.245,E2 -14426.245} C_VEL
LIN {X 0,Y 333.691,Z 216.23,A -85,B 0,C 180,E1 -14428.973,E2 -14428.973} C_VEL
LIN {X 0,Y 333.639,Z 216.24,A -85,B 0,C 180,E1 -14433.207,E2 -14433.207} C_VEL
LIN {X 0,Y 333.678,Z 216.231,A -85,B 0,C 180,E1 -14436.138,E2 -14436.138} C_VEL
LIN {X 0,Y 333.648,Z 216.238,A -85,B 0,C 180,E1 -14439.191,E2 -14439.191} C_VEL
LIN {X 0,Y 333.664,Z 216.268,A -85,B 0,C 180,E1 -14442.224,E2 -14442.224} C_VEL
LIN {X 0,Y 334.625,Z 219.074,A -85,B 0,C 180,E1 -14443.054,E2 -14443.054} C_VEL
LIN {X 0,Y 337.899,Z 226.601,A -85,B 0,C 180,E1 -14445.268,E2 -14445.268} C_VEL
LIN {X 0,Y 345.727,Z 238.646,A -85,B 0,C 180,E1 -14447.114,E2 -14447.114} C_VEL
LIN {X 0,Y 353.597,Z 251.749,A -85,B 0,C 180,E1 -14448.833,E2 -14448.833} C_VEL
LIN {X 0,Y 362.476,Z 268.584,A -85,B 0,C 180,E1 -14450.658,E2 -14450.658} C_VEL
LIN {X 0,Y 367.928,Z 280.384,A -85,B 0,C 180,E1 -14451.738,E2 -14451.738} C_VEL
LIN {X 0,Y 361.584,Z 435.599,A -85,B 0,C 180,E1 -14455.023,E2 -14455.023} C_VEL
LIN {X 0,Y 360.178,Z 451.546,A -85,B 0,C 180,E1 -14455.536,E2 -14455.536} C_VEL
LIN {X 0,Y 358.255,Z 467.712,A -85,B 0,C 180,E1 -14456.259,E2 -14456.259} C_VEL
LIN {X 0,Y 356.201,Z 482.586,A -85,B 0,C 180,E1 -14457.138,E2 -14457.138} C_VEL
LIN {X 0,Y 353.728,Z 497.385,A -85,B 0,C 180,E1 -14458.228,E2 -14458.228} C_VEL
LIN {X 0,Y 351.063,Z 511.653,A -85,B 0,C 180,E1 -14459.532,E2 -14459.532} C_VEL
LIN {X 0,Y 348.209,Z 525.326,A -85,B 0,C 180,E1 -14461.025,E2 -14461.025} C_VEL
LIN {X 0,Y 345.387,Z 538.461,A -85,B 0,C 180,E1 -14462.751,E2 -14462.751} C_VEL
LIN {X 0,Y 342.809,Z 549.7,A -85,B 0,C 180,E1 -14464.497,E2 -14464.497} C_VEL
LIN {X 0,Y 340.242,Z 560.94,A -85,B 0,C 180,E1 -14466.568,E2 -14466.568} C_VEL
LIN {X 0,Y 337.731,Z 571.854,A -85,B 0,C 180,E1 -14468.961,E2 -14468.961} C_VEL
LIN {X 0,Y 335.886,Z 581.062,A -85,B 0,C 180,E1 -14471.39,E2 -14471.39} C_VEL
LIN {X 0,Y 334.163,Z 589.641,A -85,B 0,C 180,E1 -14474.13,E2 -14474.13} C_VEL
LIN {X 0,Y 333.205,Z 595.847,A -85,B 0,C 180,E1 -14476.582,E2 -14476.582} C_VEL
LIN {X 0,Y 332.431,Z 600.876,A -85,B 0,C 180,E1 -14479.029,E2 -14479.029} C_VEL
LIN {X 0,Y 332.1,Z 604.845,A -85,B 0,C 180,E1 -14481.478,E2 -14481.478} C_VEL
LIN {X 0,Y 331.985,Z 608.018,A -85,B 0,C 180,E1 -14484.247,E2 -14484.247} C_VEL
LIN {X 0,Y 331.94,Z 609.627,A -85,B 0,C 180,E1 -14486.355,E2 -14486.355} C_VEL
LIN {X 0,Y 331.925,Z 610.486,A -85,B 0,C 180,E1 -14488.784,E2 -14488.784} C_VEL
LIN {X 0,Y 331.928,Z 610.44,A -85,B 0,C 180,E1 -14491.21,E2 -14491.21} C_VEL
LIN {X 0,Y 331.961,Z 609.331,A -85,B 0,C 180,E1 -14493.638,E2 -14493.638} C_VEL
LIN {X 0,Y 331.988,Z 607.302,A -85,B 0,C 180,E1 -14496.073,E2 -14496.073} C_VEL
LIN {X 0,Y 332.095,Z 604.153,A -85,B 0,C 180,E1 -14498.516,E2 -14498.516} C_VEL
LIN {X 0,Y 332.407,Z 600.009,A -85,B 0,C 180,E1 -14500.966,E2 -14500.966} C_VEL
LIN {X 0,Y 333.149,Z 594.649,A -85,B 0,C 180,E1 -14503.414,E2 -14503.414} C_VEL
LIN {X 0,Y 334.044,Z 588.071,A -85,B 0,C 180,E1 -14505.87,E2 -14505.87} C_VEL
LIN {X 0,Y 335.541,Z 580.164,A -85,B 0,C 180,E1 -14508.307,E2 -14508.307} C_VEL
LIN {X 0,Y 337.281,Z 570.625,A -85,B 0,C 180,E1 -14510.742,E2 -14510.742} C_VEL
LIN {X 0,Y 339.304,Z 560.751,A -85,B 0,C 180,E1 -14512.849,E2 -14512.849} C_VEL
LIN {X 0,Y 341.707,Z 549.021,A -85,B 0,C 180,E1 -14514.969,E2 -14514.969} C_VEL
LIN {X 0,Y 344.236,Z 536.655,A -85,B 0,C 180,E1 -14516.849,E2 -14516.849} C_VEL
LIN {X 0,Y 346.94,Z 522.969,A -85,B 0,C 180,E1 -14518.588,E2 -14518.588} C_VEL
LIN {X 0,Y 349.664,Z 507.913,A -85,B 0,C 180,E1 -14520.16,E2 -14520.16} C_VEL
LIN {X 0,Y 352.137,Z 493.002,A -85,B 0,C 180,E1 -14521.422,E2 -14521.422} C_VEL
LIN {X 0,Y 354.286,Z 477.831,A -85,B 0,C 180,E1 -14522.464,E2 -14522.464} C_VEL
LIN {X 0,Y 356.157,Z 461.911,A -85,B 0,C 180,E1 -14523.324,E2 -14523.324} C_VEL
LIN {X 0,Y 357.749,Z 446.198,A -85,B 0,C 180,E1 -14523.946,E2 -14523.946} C_VEL
LIN {X 0,Y 358.808,Z 428.906,A -85,B 0,C 180,E1 -14524.413,E2 -14524.413} C_VEL
LIN {X 0,Y 364.155,Z 278.715,A -85,B 0,C 180,E1 -14527.518,E2 -14527.518} C_VEL
LIN {X 0,Y 355.299,Z 260.083,A -85,B 0,C 180,E1 -14529.009,E2 -14529.009} C_VEL
LIN {X 0,Y 345.314,Z 241.09,A -85,B 0,C 180,E1 -14530.757,E2 -14530.757} C_VEL
LIN {X 0,Y 337.902,Z 227.955,A -85,B 0,C 180,E1 -14532.15,E2 -14532.15} C_VEL
LIN {X 0,Y 333.583,Z 216.238,A -85,B 0,C 180,E1 -14534.903,E2 -14534.903} C_VEL
LIN {X 0,Y 333.647,Z 216.239,A -85,B 0,C 180,E1 -14537.62,E2 -14537.62} C_VEL
LIN {X 0,Y 333.654,Z 216.24,A -85,B 0,C 180,E1 -14541.194,E2 -14541.194} C_VEL
LIN {X 0,Y 333.661,Z 216.235,A -85,B 0,C 180,E1 -14545.224,E2 -14545.224} C_VEL
LIN {X 0,Y 333.603,Z 216.221,A -85,B 0,C 180,E1 -14548.22,E2 -14548.22} C_VEL
LIN {X 0,Y 333.661,Z 216.239,A -85,B 0,C 180,E1 -14551.024,E2 -14551.024} C_VEL
LIN {X 0,Y 333.708,Z 216.205,A -85,B 0,C 180,E1 -14553.752,E2 -14553.752} C_VEL
LIN {X 0,Y 333.694,Z 216.229,A -85,B 0,C 180,E1 -14557.912,E2 -14557.912} C_VEL
LIN {X 0,Y 333.766,Z 216.203,A -85,B 0,C 180,E1 -14561.589,E2 -14561.589} C_VEL
LIN {X 0,Y 333.779,Z 216.21,A -85,B 0,C 180,E1 -14565.576,E2 -14565.576} C_VEL
LIN {X 0,Y 333.807,Z 216.188,A -85,B 0,C 180,E1 -14569.078,E2 -14569.078} C_VEL
LIN {X 0,Y 333.986,Z 216.192,A -85,B 0,C 180,E1 -14572.747,E2 -14572.747} C_VEL
LIN {X 0,Y 333.782,Z 216.187,A -85,B 0,C 180,E1 -14575.169,E2 -14575.169} C_VEL
LIN {X 0,Y 334.076,Z 216.151,A -85,B 0,C 180,E1 -14577.589,E2 -14577.589} C_VEL
LIN {X 0,Y 334.218,Z 216.162,A -85,B 0,C 180,E1 -14580.001,E2 -14580.001} C_VEL
LIN {X 0,Y 334.076,Z 216.177,A -85,B 0,C 180,E1 -14582.412,E2 -14582.412} C_VEL
LIN {X 0,Y 333.962,Z 216.188,A -85,B 0,C 180,E1 -14586.71,E2 -14586.71} C_VEL
LIN {X 0,Y 333.822,Z 216.208,A -85,B 0,C 180,E1 -14589.697,E2 -14589.697} C_VEL
LIN {X 0,Y 333.768,Z 216.211,A -85,B 0,C 180,E1 -14593.393,E2 -14593.393} C_VEL
LIN {X 0,Y 333.72,Z 216.215,A -85,B 0,C 180,E1 -14597.148,E2 -14597.148} C_VEL
LIN {X 0,Y 333.712,Z 216.207,A -85,B 0,C 180,E1 -14599.693,E2 -14599.693} C_VEL
LIN {X 0,Y 333.667,Z 216.234,A -85,B 0,C 180,E1 -14602.281,E2 -14602.281} C_VEL
LIN {X 0,Y 333.711,Z 216.205,A -85,B 0,C 180,E1 -14606.249,E2 -14606.249} C_VEL
LIN {X 0,Y 333.687,Z 216.232,A -85,B 0,C 180,E1 -14608.975,E2 -14608.975} C_VEL
LIN {X 0,Y 333.621,Z 216.218,A -85,B 0,C 180,E1 -14612.59,E2 -14612.59} C_VEL
LIN {X 0,Y 333.655,Z 216.238,A -85,B 0,C 180,E1 -14616.142,E2 -14616.142} C_VEL
LIN {X 0,Y 333.627,Z 216.217,A -85,B 0,C 180,E1 -14619.196,E2 -14619.196} C_VEL
LIN {X 0,Y 333.615,Z 216.242,A -85,B 0,C 180,E1 -14622.503,E2 -14622.503} C_VEL
LIN {X 0,Y 333.58,Z 216.229,A -85,B 0,C 180,E1 -14625.958,E2 -14625.958} C_VEL
LIN {X 0,Y 333.629,Z 216.234,A -85,B 0,C 180,E1 -14629.32,E2 -14629.32} C_VEL
LIN {X 0,Y 333.652,Z 216.236,A -85,B 0,C 180,E1 -14633.172,E2 -14633.172} C_VEL
LIN {X 0,Y 333.664,Z 216.22,A -85,B 0,C 180,E1 -14635.345,E2 -14635.345} C_VEL
LIN {X 0,Y 333.621,Z 216.241,A -85,B 0,C 180,E1 -14638.226,E2 -14638.226} C_VEL
LIN {X 0,Y 333.647,Z 216.231,A -85,B 0,C 180,E1 -14641.026,E2 -14641.026} C_VEL
LIN {X 0,Y 333.691,Z 216.227,A -85,B 0,C 180,E1 -14645.092,E2 -14645.092} C_VEL
LIN {X 0,Y 333.66,Z 216.237,A -85,B 0,C 180,E1 -14649.022,E2 -14649.022} C_VEL
LIN {X 0,Y 333.738,Z 216.223,A -85,B 0,C 180,E1 -14651.59,E2 -14651.59} C_VEL
LIN {X 0,Y 333.764,Z 216.223,A -85,B 0,C 180,E1 -14654.472,E2 -14654.472} C_VEL
LIN {X 0,Y 334.704,Z 218.955,A -85,B 0,C 180,E1 -14654.688,E2 -14654.688} C_VEL
LIN {X 0,Y 336.65,Z 221.609,A -85,B 0,C 180,E1 -14655.039,E2 -14655.039} C_VEL
LIN {X 0,Y 348.346,Z 240.111,A -85,B 0,C 180,E1 -14657.107,E2 -14657.107} C_VEL
LIN {X 0,Y 354.348,Z 250.566,A -85,B 0,C 180,E1 -14658.129,E2 -14658.129} C_VEL
LIN {X 0,Y 360.933,Z 263.632,A -85,B 0,C 180,E1 -14659.236,E2 -14659.236} C_VEL
LIN {X 0,Y 364.23,Z 271.117,A -85,B 0,C 180,E1 -14659.795,E2 -14659.795} C_VEL
LIN {X 0,Y 358.781,Z 418.906,A -85,B 0,C 180,E1 -14662.865,E2 -14662.865} C_VEL
LIN {X 0,Y 357.543,Z 435.976,A -85,B 0,C 180,E1 -14663.442,E2 -14663.442} C_VEL
LIN {X 0,Y 355.958,Z 451.795,A -85,B 0,C 180,E1 -14664.195,E2 -14664.195} C_VEL
LIN {X 0,Y 354.054,Z 467.399,A -85,B 0,C 180,E1 -14665.164,E2 -14665.164} C_VEL
LIN {X 0,Y 351.844,Z 482.924,A -85,B 0,C 180,E1 -14666.378,E2 -14666.378} C_VEL
LIN {X 0,Y 349.467,Z 496.878,A -85,B 0,C 180,E1 -14667.698,E2 -14667.698} C_VEL
LIN {X 0,Y 346.963,Z 510.553,A -85,B 0,C 180,E1 -14669.277,E2 -14669.277} C_VEL
LIN {X 0,Y 344.427,Z 522.981,A -85,B 0,C 180,E1 -14670.979,E2 -14670.979} C_VEL
LIN {X 0,Y 341.985,Z 535.053,A -85,B 0,C 180,E1 -14672.948,E2 -14672.948} C_VEL
LIN {X 0,Y 339.717,Z 545.659,A -85,B 0,C 180,E1 -14674.983,E2 -14674.983} C_VEL
LIN {X 0,Y 337.676,Z 555.214,A -85,B 0,C 180,E1 -14677.176,E2 -14677.176} C_VEL
LIN {X 0,Y 335.846,Z 564.206,A -85,B 0,C 180,E1 -14679.64,E2 -14679.64} C_VEL
LIN {X 0,Y 334.478,Z 571.719,A -85,B 0,C 180,E1 -14682.132,E2 -14682.132} C_VEL
LIN {X 0,Y 333.41,Z 577.953,A -85,B 0,C 180,E1 -14684.655,E2 -14684.655} C_VEL
LIN {X 0,Y 332.679,Z 582.883,A -85,B 0,C 180,E1 -14687.205,E2 -14687.205} C_VEL
LIN {X 0,Y 332.156,Z 586.714,A -85,B 0,C 180,E1 -14689.79,E2 -14689.79} C_VEL
LIN {X 0,Y 331.767,Z 589.459,A -85,B 0,C 180,E1 -14692.417,E2 -14692.417} C_VEL
LIN {X 0,Y 331.64,Z 590.678,A -85,B 0,C 180,E1 -14694.299,E2 -14694.299} C_VEL
LIN {X 0,Y 330.957,Z 591.154,A -85,B 0,C 180,E1 -14695.309,E2 -14695.309} C_VEL
LIN {X 0,Y 328.066,Z 591.533,A -85,B 0,C 180,E1 -14696.957,E2 -14696.957} C_VEL
LIN {X 0,Y 325.658,Z 591.554,A -85,B 0,C 180,E1 -14698.294,E2 -14698.294} C_VEL
LIN {X 0,Y 324.678,Z 591.391,A -85,B 0,C 180,E1 -14699.328,E2 -14699.328} C_VEL
LIN {X 0,Y 324.627,Z 591.244,A -85,B 0,C 180,E1 -14699.678,E2 -14699.678} C_VEL
LIN {X 0,Y 324.829,Z 589.757,A -85,B 0,C 180,E1 -14702.455,E2 -14702.455} C_VEL
LIN {X 0,Y 325.198,Z 587.483,A -85,B 0,C 180,E1 -14704.79,E2 -14704.79} C_VEL
LIN {X 0,Y 325.781,Z 584.351,A -85,B 0,C 180,E1 -14707.162,E2 -14707.162} C_VEL
LIN {X 0,Y 326.818,Z 578.909,A -85,B 0,C 180,E1 -14710.177,E2 -14710.177} C_VEL
LIN {X 0,Y 327.875,Z 573.64,A -85,B 0,C 180,E1 -14712.472,E2 -14712.472} C_VEL
LIN {X 0,Y 329.68,Z 565.708,A -85,B 0,C 180,E1 -14715.292,E2 -14715.292} C_VEL
LIN {X 0,Y 331.877,Z 556.916,A -85,B 0,C 180,E1 -14717.834,E2 -14717.834} C_VEL
LIN {X 0,Y 334.253,Z 547.338,A -85,B 0,C 180,E1 -14720.127,E2 -14720.127} C_VEL
LIN {X 0,Y 336.835,Z 536.962,A -85,B 0,C 180,E1 -14722.214,E2 -14722.214} C_VEL
LIN {X 0,Y 339.684,Z 525.338,A -85,B 0,C 180,E1 -14724.191,E2 -14724.191} C_VEL
LIN {X 0,Y 342.498,Z 513.335,A -85,B 0,C 180,E1 -14725.92,E2 -14725.92} C_VEL
LIN {X 0,Y 345.476,Z 499.371,A -85,B 0,C 180,E1 -14727.591,E2 -14727.591} C_VEL
LIN {X 0,Y 348.146,Z 485.653,A -85,B 0,C 180,E1 -14728.948,E2 -14728.948} C_VEL
LIN {X 0,Y 350.703,Z 470.839,A -85,B 0,C 180,E1 -14730.153,E2 -14730.153} C_VEL
LIN {X 0,Y 352.953,Z 455.131,A -85,B 0,C 180,E1 -14731.18,E2 -14731.18} C_VEL
LIN {X 0,Y 354.82,Z 438.85,A -85,B 0,C 180,E1 -14731.995,E2 -14731.995} C_VEL
LIN {X 0,Y 356.231,Z 421.894,A -85,B 0,C 180,E1 -14732.599,E2 -14732.599} C_VEL
LIN {X 0,Y 357.454,Z 395.616,A -85,B 0,C 180,E1 -14733.208,E2 -14733.208} C_VEL
LIN {X 0,Y 362.721,Z 275.405,A -85,B 0,C 180,E1 -14735.755,E2 -14735.755} C_VEL
LIN {X 0,Y 354.371,Z 258.944,A -85,B 0,C 180,E1 -14737.469,E2 -14737.469} C_VEL
LIN {X 0,Y 347.516,Z 247.22,A -85,B 0,C 180,E1 -14738.943,E2 -14738.943} C_VEL
LIN {X 0,Y 339.573,Z 235.56,A -85,B 0,C 180,E1 -14740.744,E2 -14740.744} C_VEL
LIN {X 0,Y 336.146,Z 230.877,A -85,B 0,C 180,E1 -14741.568,E2 -14741.568} C_VEL
LIN {X 0,Y 333.201,Z 226.691,A -85,B 0,C 180,E1 -14742.31,E2 -14742.31} C_VEL
LIN {X 0,Y 330.822,Z 223.566,A -85,B 0,C 180,E1 -14742.919,E2 -14742.919} C_VEL
LIN {X 0,Y 329.969,Z 222.203,A -85,B 0,C 180,E1 -14743.153,E2 -14743.153} C_VEL
LIN {X 0,Y 327.887,Z 220.175,A -85,B 0,C 180,E1 -14743.688,E2 -14743.688} C_VEL
LIN {X 0,Y 326.858,Z 217.828,A -85,B 0,C 180,E1 -14744.008,E2 -14744.008} C_VEL
LIN {X 0,Y 326.735,Z 217.098,A -85,B 0,C 180,E1 -14744.082,E2 -14744.082} C_VEL
LIN {X 0,Y 326.736,Z 217.096,A -85,B 0,C 180,E1 -14747.578,E2 -14747.578} C_VEL
LIN {X 0,Y 326.904,Z 217.074,A -85,B 0,C 180,E1 -14751.474,E2 -14751.474} C_VEL
LIN {X 0,Y 326.991,Z 217.062,A -85,B 0,C 180,E1 -14753.83,E2 -14753.83} C_VEL
LIN {X 0,Y 327.046,Z 217.06,A -85,B 0,C 180,E1 -14757.536,E2 -14757.536} C_VEL
LIN {X 0,Y 327.163,Z 217.044,A -85,B 0,C 180,E1 -14759.999,E2 -14759.999} C_VEL
LIN {X 0,Y 327.046,Z 217.057,A -85,B 0,C 180,E1 -14762.463,E2 -14762.463} C_VEL
LIN {X 0,Y 326.96,Z 217.07,A -85,B 0,C 180,E1 -14766.169,E2 -14766.169} C_VEL
LIN {X 0,Y 326.786,Z 217.086,A -85,B 0,C 180,E1 -14769.906,E2 -14769.906} C_VEL
LIN {X 0,Y 326.759,Z 217.091,A -85,B 0,C 180,E1 -14773.685,E2 -14773.685} C_VEL
LIN {X 0,Y 326.667,Z 217.109,A -85,B 0,C 180,E1 -14777.529,E2 -14777.529} C_VEL
LIN {X 0,Y 326.621,Z 217.107,A -85,B 0,C 180,E1 -14781.456,E2 -14781.456} C_VEL
LIN {X 0,Y 326.693,Z 217.103,A -85,B 0,C 180,E1 -14785.483,E2 -14785.483} C_VEL
LIN {X 0,Y 326.653,Z 217.109,A -85,B 0,C 180,E1 -14788.25,E2 -14788.25} C_VEL
LIN {X 0,Y 326.578,Z 217.118,A -85,B 0,C 180,E1 -14791.096,E2 -14791.096} C_VEL
LIN {X 0,Y 326.609,Z 217.11,A -85,B 0,C 180,E1 -14794.018,E2 -14794.018} C_VEL
LIN {X 0,Y 326.629,Z 217.112,A -85,B 0,C 180,E1 -14797.237,E2 -14797.237} C_VEL
LIN {X 0,Y 326.621,Z 217.259,A -85,B 0,C 180,E1 -14800.872,E2 -14800.872} C_VEL
LIN {X 0,Y 328.124,Z 220.621,A -85,B 0,C 180,E1 -14802.015,E2 -14802.015} C_VEL
LIN {X 0,Y 330.416,Z 226.32,A -85,B 0,C 180,E1 -14803.73,E2 -14803.73} C_VEL
LIN {X 0,Y 335.8,Z 234.306,A -85,B 0,C 180,E1 -14805.118,E2 -14805.118} C_VEL
LIN {X 0,Y 341.743,Z 243.496,A -85,B 0,C 180,E1 -14806.555,E2 -14806.555} C_VEL
LIN {X 0,Y 349.546,Z 256.705,A -85,B 0,C 180,E1 -14808.325,E2 -14808.325} C_VEL
LIN {X 0,Y 356.824,Z 270.652,A -85,B 0,C 180,E1 -14809.885,E2 -14809.885} C_VEL
LIN {X 0,Y 362.479,Z 282.686,A -85,B 0,C 180,E1 -14811.047,E2 -14811.047} C_VEL
LIN {X 0,Y 357.437,Z 400.165,A -85,B 0,C 180,E1 -14813.545,E2 -14813.545} C_VEL
LIN {X 0,Y 355.862,Z 436.704,A -85,B 0,C 180,E1 -14814.369,E2 -14814.369} C_VEL
LIN {X 0,Y 354.393,Z 452.481,A -85,B 0,C 180,E1 -14814.891,E2 -14814.891} C_VEL
LIN {X 0,Y 352.416,Z 468.315,A -85,B 0,C 180,E1 -14815.622,E2 -14815.622} C_VEL
LIN {X 0,Y 350.264,Z 482.998,A -85,B 0,C 180,E1 -14816.509,E2 -14816.509} C_VEL
LIN {X 0,Y 347.727,Z 497.721,A -85,B 0,C 180,E1 -14817.614,E2 -14817.614} C_VEL
LIN {X 0,Y 344.944,Z 511.891,A -85,B 0,C 180,E1 -14818.932,E2 -14818.932} C_VEL
LIN {X 0,Y 341.968,Z 525.458,A -85,B 0,C 180,E1 -14820.444,E2 -14820.444} C_VEL
LIN {X 0,Y 339.035,Z 538.509,A -85,B 0,C 180,E1 -14822.196,E2 -14822.196} C_VEL
LIN {X 0,Y 336.036,Z 551.063,A -85,B 0,C 180,E1 -14824.2,E2 -14824.2} C_VEL
LIN {X 0,Y 333.305,Z 562.421,A -85,B 0,C 180,E1 -14826.38,E2 -14826.38} C_VEL
LIN {X 0,Y 331.009,Z 571.806,A -85,B 0,C 180,E1 -14828.513,E2 -14828.513} C_VEL
LIN {X 0,Y 329.049,Z 580.977,A -85,B 0,C 180,E1 -14830.989,E2 -14830.989} C_VEL
LIN {X 0,Y 327.222,Z 589.52,A -85,B 0,C 180,E1 -14833.784,E2 -14833.784} C_VEL
LIN {X 0,Y 326.199,Z 595.717,A -85,B 0,C 180,E1 -14836.288,E2 -14836.288} C_VEL
LIN {X 0,Y 325.41,Z 600.727,A -85,B 0,C 180,E1 -14838.789,E2 -14838.789} C_VEL
LIN {X 0,Y 325.029,Z 604.688,A -85,B 0,C 180,E1 -14841.292,E2 -14841.292} C_VEL
LIN {X 0,Y 324.889,Z 608.014,A -85,B 0,C 180,E1 -14844.305,E2 -14844.305} C_VEL
LIN {X 0,Y 324.846,Z 609.444,A -85,B 0,C 180,E1 -14846.276,E2 -14846.276} C_VEL
LIN {X 0,Y 324.833,Z 610.285,A -85,B 0,C 180,E1 -14848.757,E2 -14848.757} C_VEL
LIN {X 0,Y 324.836,Z 610.23,A -85,B 0,C 180,E1 -14851.237,E2 -14851.237} C_VEL
LIN {X 0,Y 324.864,Z 609.102,A -85,B 0,C 180,E1 -14853.718,E2 -14853.718} C_VEL
LIN {X 0,Y 324.887,Z 607.061,A -85,B 0,C 180,E1 -14856.206,E2 -14856.206} C_VEL
LIN {X 0,Y 325.024,Z 603.892,A -85,B 0,C 180,E1 -14858.702,E2 -14858.702} C_VEL
LIN {X 0,Y 325.386,Z 599.723,A -85,B 0,C 180,E1 -14861.206,E2 -14861.206} C_VEL
LIN {X 0,Y 326.152,Z 594.345,A -85,B 0,C 180,E1 -14863.708,E2 -14863.708} C_VEL
LIN {X 0,Y 327.127,Z 587.736,A -85,B 0,C 180,E1 -14866.214,E2 -14866.214} C_VEL
LIN {X 0,Y 328.662,Z 579.794,A -85,B 0,C 180,E1 -14868.705,E2 -14868.705} C_VEL
LIN {X 0,Y 330.515,Z 570.237,A -85,B 0,C 180,E1 -14871.187,E2 -14871.187} C_VEL
LIN {X 0,Y 332.966,Z 558.814,A -85,B 0,C 180,E1 -14873.639,E2 -14873.639} C_VEL
LIN {X 0,Y 335.449,Z 547.148,A -85,B 0,C 180,E1 -14875.726,E2 -14875.726} C_VEL
LIN {X 0,Y 338.064,Z 535.048,A -85,B 0,C 180,E1 -14877.548,E2 -14877.548} C_VEL
LIN {X 0,Y 340.607,Z 522.38,A -85,B 0,C 180,E1 -14879.17,E2 -14879.17} C_VEL
LIN {X 0,Y 343.478,Z 507.276,A -85,B 0,C 180,E1 -14880.761,E2 -14880.761} C_VEL
LIN {X 0,Y 346.052,Z 492.262,A -85,B 0,C 180,E1 -14882.04,E2 -14882.04} C_VEL
LIN {X 0,Y 348.26,Z 476.923,A -85,B 0,C 180,E1 -14883.097,E2 -14883.097} C_VEL
LIN {X 0,Y 350.271,Z 459.981,A -85,B 0,C 180,E1 -14884.002,E2 -14884.002} C_VEL
LIN {X 0,Y 351.911,Z 443.503,A -85,B 0,C 180,E1 -14884.631,E2 -14884.631} C_VEL
LIN {X 0,Y 352.934,Z 426.492,A -85,B 0,C 180,E1 -14885.074,E2 -14885.074} C_VEL
LIN {X 0,Y 358.304,Z 280.981,A -85,B 0,C 180,E1 -14888.123,E2 -14888.123} C_VEL
LIN {X 0,Y 349.765,Z 262.917,A -85,B 0,C 180,E1 -14889.606,E2 -14889.606} C_VEL
LIN {X 0,Y 338.524,Z 241.714,A -85,B 0,C 180,E1 -14891.636,E2 -14891.636} C_VEL
LIN {X 0,Y 330.482,Z 227.707,A -85,B 0,C 180,E1 -14893.212,E2 -14893.212} C_VEL
LIN {X 0,Y 326.541,Z 217.111,A -85,B 0,C 180,E1 -14895.775,E2 -14895.775} C_VEL
LIN {X 0,Y 326.568,Z 217.107,A -85,B 0,C 180,E1 -14898.864,E2 -14898.864} C_VEL
LIN {X 0,Y 326.62,Z 217.114,A -85,B 0,C 180,E1 -14901.392,E2 -14901.392} C_VEL
LIN {X 0,Y 326.595,Z 217.11,A -85,B 0,C 180,E1 -14904.849,E2 -14904.849} C_VEL
LIN {X 0,Y 326.582,Z 217.098,A -85,B 0,C 180,E1 -14907.453,E2 -14907.453} C_VEL
LIN {X 0,Y 326.62,Z 217.113,A -85,B 0,C 180,E1 -14910.338,E2 -14910.338} C_VEL
LIN {X 0,Y 326.664,Z 217.086,A -85,B 0,C 180,E1 -14914.515,E2 -14914.515} C_VEL
LIN {X 0,Y 326.638,Z 217.096,A -85,B 0,C 180,E1 -14918.545,E2 -14918.545} C_VEL
LIN {X 0,Y 326.717,Z 217.074,A -85,B 0,C 180,E1 -14921.176,E2 -14921.176} C_VEL
LIN {X 0,Y 326.734,Z 217.088,A -85,B 0,C 180,E1 -14925.433,E2 -14925.433} C_VEL
LIN {X 0,Y 326.743,Z 217.063,A -85,B 0,C 180,E1 -14928.839,E2 -14928.839} C_VEL
LIN {X 0,Y 326.939,Z 217.072,A -85,B 0,C 180,E1 -14932.59,E2 -14932.59} C_VEL
LIN {X 0,Y 326.748,Z 217.063,A -85,B 0,C 180,E1 -14935.065,E2 -14935.065} C_VEL
LIN {X 0,Y 327.017,Z 217.028,A -85,B 0,C 180,E1 -14937.537,E2 -14937.537} C_VEL
LIN {X 0,Y 327.169,Z 217.04,A -85,B 0,C 180,E1 -14940.001,E2 -14940.001} C_VEL
LIN {X 0,Y 327.017,Z 217.055,A -85,B 0,C 180,E1 -14942.464,E2 -14942.464} C_VEL
LIN {X 0,Y 326.928,Z 217.063,A -85,B 0,C 180,E1 -14946.703,E2 -14946.703} C_VEL
LIN {X 0,Y 326.777,Z 217.082,A -85,B 0,C 180,E1 -14949.908,E2 -14949.908} C_VEL
LIN {X 0,Y 326.731,Z 217.089,A -85,B 0,C 180,E1 -14953.687,E2 -14953.687} C_VEL
LIN {X 0,Y 326.672,Z 217.091,A -85,B 0,C 180,E1 -14957.53,E2 -14957.53} C_VEL
LIN {X 0,Y 326.639,Z 217.091,A -85,B 0,C 180,E1 -14960.137,E2 -14960.137} C_VEL
LIN {X 0,Y 326.627,Z 217.101,A -85,B 0,C 180,E1 -14964.132,E2 -14964.132} C_VEL
LIN {X 0,Y 326.66,Z 217.087,A -85,B 0,C 180,E1 -14966.861,E2 -14966.861} C_VEL
LIN {X 0,Y 326.617,Z 217.107,A -85,B 0,C 180,E1 -14970.614,E2 -14970.614} C_VEL
LIN {X 0,Y 326.586,Z 217.101,A -85,B 0,C 180,E1 -14974.023,E2 -14974.023} C_VEL
LIN {X 0,Y 326.607,Z 217.11,A -85,B 0,C 180,E1 -14977.242,E2 -14977.242} C_VEL
LIN {X 0,Y 326.56,Z 217.117,A -85,B 0,C 180,E1 -14981.135,E2 -14981.135} C_VEL
LIN {X 0,Y 326.51,Z 217.107,A -85,B 0,C 180,E1 -14984.746,E2 -14984.746} C_VEL
LIN {X 0,Y 326.56,Z 217.122,A -85,B 0,C 180,E1 -14988.158,E2 -14988.158} C_VEL
LIN {X 0,Y 326.574,Z 217.107,A -85,B 0,C 180,E1 -14991.39,E2 -14991.39} C_VEL
LIN {X 0,Y 326.608,Z 217.101,A -85,B 0,C 180,E1 -14994.855,E2 -14994.855} C_VEL
LIN {X 0,Y 326.599,Z 217.114,A -85,B 0,C 180,E1 -14997.459,E2 -14997.459} C_VEL
LIN {X 0,Y 326.609,Z 217.102,A -85,B 0,C 180,E1 -15000.341,E2 -15000.341} C_VEL
LIN {X 0,Y 326.636,Z 217.102,A -85,B 0,C 180,E1 -15004.648,E2 -15004.648} C_VEL
LIN {X 0,Y 326.611,Z 217.11,A -85,B 0,C 180,E1 -15008.547,E2 -15008.547} C_VEL
LIN {X 0,Y 326.651,Z 217.111,A -85,B 0,C 180,E1 -15012.473,E2 -15012.473} C_VEL
LIN {X 0,Y 326.665,Z 217.102,A -85,B 0,C 180,E1 -15013.441,E2 -15013.441} C_VEL
LIN {X 0,Y 327.713,Z 220.046,A -85,B 0,C 180,E1 -15013.695,E2 -15013.695} C_VEL
LIN {X 0,Y 329.626,Z 222.473,A -85,B 0,C 180,E1 -15014.053,E2 -15014.053} C_VEL
LIN {X 0,Y 337.541,Z 234.747,A -85,B 0,C 180,E1 -15015.535,E2 -15015.535} C_VEL
LIN {X 0,Y 347.884,Z 251.705,A -85,B 0,C 180,E1 -15017.359,E2 -15017.359} C_VEL
LIN {X 0,Y 355.834,Z 267.511,A -85,B 0,C 180,E1 -15018.744,E2 -15018.744} C_VEL
LIN {X 0,Y 358.329,Z 272.949,A -85,B 0,C 180,E1 -15019.173,E2 -15019.173} C_VEL
LIN {X 0,Y 352.824,Z 418.386,A -85,B 0,C 180,E1 -15022.24,E2 -15022.24} C_VEL
LIN {X 0,Y 351.516,Z 435.747,A -85,B 0,C 180,E1 -15022.825,E2 -15022.825} C_VEL
LIN {X 0,Y 349.896,Z 451.677,A -85,B 0,C 180,E1 -15023.588,E2 -15023.588} C_VEL
LIN {X 0,Y 348.069,Z 466.378,A -85,B 0,C 180,E1 -15024.499,E2 -15024.499} C_VEL
LIN {X 0,Y 345.908,Z 481.348,A -85,B 0,C 180,E1 -15025.657,E2 -15025.657} C_VEL
LIN {X 0,Y 343.332,Z 496.215,A -85,B 0,C 180,E1 -15027.07,E2 -15027.07} C_VEL
LIN {X 0,Y 340.707,Z 510.052,A -85,B 0,C 180,E1 -15028.673,E2 -15028.673} C_VEL
LIN {X 0,Y 338.077,Z 522.512,A -85,B 0,C 180,E1 -15030.388,E2 -15030.388} C_VEL
LIN {X 0,Y 335.484,Z 534.779,A -85,B 0,C 180,E1 -15032.404,E2 -15032.404} C_VEL
LIN {X 0,Y 333.058,Z 545.749,A -85,B 0,C 180,E1 -15034.541,E2 -15034.541} C_VEL
LIN {X 0,Y 330.697,Z 556.315,A -85,B 0,C 180,E1 -15037.022,E2 -15037.022} C_VEL
LIN {X 0,Y 328.841,Z 565.144,A -85,B 0,C 180,E1 -15039.537,E2 -15039.537} C_VEL
LIN {X 0,Y 327.555,Z 571.69,A -85,B 0,C 180,E1 -15041.764,E2 -15041.764} C_VEL
LIN {X 0,Y 326.438,Z 577.962,A -85,B 0,C 180,E1 -15044.342,E2 -15044.342} C_VEL
LIN {X 0,Y 325.668,Z 582.924,A -85,B 0,C 180,E1 -15046.94,E2 -15046.94} C_VEL
LIN {X 0,Y 325.241,Z 585.952,A -85,B 0,C 180,E1 -15048.915,E2 -15048.915} C_VEL
LIN {X 0,Y 324.81,Z 588.956,A -85,B 0,C 180,E1 -15051.584,E2 -15051.584} C_VEL
LIN {X 0,Y 324.53,Z 590.996,A -85,B 0,C 180,E1 -15054.555,E2 -15054.555} C_VEL
LIN {X 0,Y 324.561,Z 591.685,A -85,B 0,C 180,E1 -15057.399,E2 -15057.399} C_VEL
LIN {X 0,Y 324.627,Z 591.244,A -85,B 0,C 180,E1 -15059.678,E2 -15059.678} C_VEL
LIN {X 0,Y 324.056,Z 590.896,A -85,B 0,C 180,E1 -15060.713,E2 -15060.713} C_VEL
LIN {X 0,Y 321.343,Z 589.979,A -85,B 0,C 180,E1 -15062.399,E2 -15062.399} C_VEL
LIN {X 0,Y 319.07,Z 588.922,A -85,B 0,C 180,E1 -15063.757,E2 -15063.757} C_VEL
LIN {X 0,Y 318.187,Z 587.92,A -85,B 0,C 180,E1 -15064.8,E2 -15064.8} C_VEL
LIN {X 0,Y 318.168,Z 587.528,A -85,B 0,C 180,E1 -15065.151,E2 -15065.151} C_VEL
LIN {X 0,Y 318.954,Z 583.479,A -85,B 0,C 180,E1 -15068.097,E2 -15068.097} C_VEL
LIN {X 0,Y 319.842,Z 579.323,A -85,B 0,C 180,E1 -15070.408,E2 -15070.408} C_VEL
LIN {X 0,Y 320.947,Z 574.113,A -85,B 0,C 180,E1 -15072.754,E2 -15072.754} C_VEL
LIN {X 0,Y 322.729,Z 566.718,A -85,B 0,C 180,E1 -15075.483,E2 -15075.483} C_VEL
LIN {X 0,Y 324.794,Z 558.776,A -85,B 0,C 180,E1 -15077.871,E2 -15077.871} C_VEL
LIN {X 0,Y 327.138,Z 549.856,A -85,B 0,C 180,E1 -15080.128,E2 -15080.128} C_VEL
LIN {X 0,Y 329.537,Z 540.768,A -85,B 0,C 180,E1 -15082.103,E2 -15082.103} C_VEL
LIN {X 0,Y 332.516,Z 529.22,A -85,B 0,C 180,E1 -15084.204,E2 -15084.204} C_VEL
LIN {X 0,Y 335.655,Z 516.455,A -85,B 0,C 180,E1 -15086.149,E2 -15086.149} C_VEL
LIN {X 0,Y 338.801,Z 502.82,A -85,B 0,C 180,E1 -15087.875,E2 -15087.875} C_VEL
LIN {X 0,Y 341.594,Z 489.506,A -85,B 0,C 180,E1 -15089.282,E2 -15089.282} C_VEL
LIN {X 0,Y 344.216,Z 475.042,A -85,B 0,C 180,E1 -15090.545,E2 -15090.545} C_VEL
LIN {X 0,Y 346.605,Z 460.157,A -85,B 0,C 180,E1 -15091.584,E2 -15091.584} C_VEL
LIN {X 0,Y 348.729,Z 443.356,A -85,B 0,C 180,E1 -15092.507,E2 -15092.507} C_VEL
LIN {X 0,Y 350.336,Z 426.607,A -85,B 0,C 180,E1 -15093.177,E2 -15093.177} C_VEL
LIN {X 0,Y 351.473,Z 409.393,A -85,B 0,C 180,E1 -15093.629,E2 -15093.629} C_VEL
LIN {X 0,Y 357.337,Z 277.909,A -85,B 0,C 180,E1 -15096.465,E2 -15096.465} C_VEL
LIN {X 0,Y 349.78,Z 262.977,A -85,B 0,C 180,E1 -15098.081,E2 -15098.081} C_VEL
LIN {X 0,Y 343.683,Z 252.401,A -85,B 0,C 180,E1 -15099.446,E2 -15099.446} C_VEL
LIN {X 0,Y 335.895,Z 240.805,A -85,B 0,C 180,E1 -15101.276,E2 -15101.276} C_VEL
LIN {X 0,Y 329.634,Z 232.092,A -85,B 0,C 180,E1 -15102.863,E2 -15102.863} C_VEL
LIN {X 0,Y 326.633,Z 227.968,A -85,B 0,C 180,E1 -15103.676,E2 -15103.676} C_VEL
LIN {X 0,Y 324.27,Z 225.164,A -85,B 0,C 180,E1 -15104.321,E2 -15104.321} C_VEL
LIN {X 0,Y 323.247,Z 223.28,A -85,B 0,C 180,E1 -15104.634,E2 -15104.634} C_VEL
LIN {X 0,Y 320.954,Z 221.156,A -85,B 0,C 180,E1 -15105.274,E2 -15105.274} C_VEL
LIN {X 0,Y 319.848,Z 218.591,A -85,B 0,C 180,E1 -15105.652,E2 -15105.652} C_VEL
LIN {X 0,Y 319.732,Z 217.969,A -85,B 0,C 180,E1 -15105.745,E2 -15105.745} C_VEL
LIN {X 0,Y 319.741,Z 217.967,A -85,B 0,C 180,E1 -15109.872,E2 -15109.872} C_VEL
LIN {X 0,Y 319.946,Z 217.94,A -85,B 0,C 180,E1 -15113.694,E2 -15113.694} C_VEL
LIN {X 0,Y 319.99,Z 217.938,A -85,B 0,C 180,E1 -15117.482,E2 -15117.482} C_VEL
LIN {X 0,Y 320.116,Z 217.922,A -85,B 0,C 180,E1 -15119.999,E2 -15119.999} C_VEL
LIN {X 0,Y 319.99,Z 217.936,A -85,B 0,C 180,E1 -15122.517,E2 -15122.517} C_VEL
LIN {X 0,Y 319.916,Z 217.947,A -85,B 0,C 180,E1 -15126.306,E2 -15126.306} C_VEL
LIN {X 0,Y 319.738,Z 217.963,A -85,B 0,C 180,E1 -15130.127,E2 -15130.127} C_VEL
LIN {X 0,Y 319.734,Z 217.968,A -85,B 0,C 180,E1 -15133.991,E2 -15133.991} C_VEL
LIN {X 0,Y 319.617,Z 217.984,A -85,B 0,C 180,E1 -15137.929,E2 -15137.929} C_VEL
LIN {X 0,Y 319.571,Z 217.985,A -85,B 0,C 180,E1 -15141.953,E2 -15141.953} C_VEL
LIN {X 0,Y 319.637,Z 217.982,A -85,B 0,C 180,E1 -15146.087,E2 -15146.087} C_VEL
LIN {X 0,Y 319.575,Z 217.988,A -85,B 0,C 180,E1 -15148.934,E2 -15148.934} C_VEL
LIN {X 0,Y 319.528,Z 217.991,A -85,B 0,C 180,E1 -15151.862,E2 -15151.862} C_VEL
LIN {X 0,Y 319.582,Z 217.99,A -85,B 0,C 180,E1 -15155.541,E2 -15155.541} C_VEL
LIN {X 0,Y 319.576,Z 218.004,A -85,B 0,C 180,E1 -15159.318,E2 -15159.318} C_VEL
LIN {X 0,Y 320.564,Z 220.849,A -85,B 0,C 180,E1 -15160.296,E2 -15160.296} C_VEL
LIN {X 0,Y 322.87,Z 225.782,A -85,B 0,C 180,E1 -15162.01,E2 -15162.01} C_VEL
LIN {X 0,Y 331.512,Z 238.437,A -85,B 0,C 180,E1 -15164.394,E2 -15164.394} C_VEL
LIN {X 0,Y 338.23,Z 249.077,A -85,B 0,C 180,E1 -15166.088,E2 -15166.088} C_VEL
LIN {X 0,Y 345.559,Z 261.67,A -85,B 0,C 180,E1 -15167.808,E2 -15167.808} C_VEL
LIN {X 0,Y 353.397,Z 277.043,A -85,B 0,C 180,E1 -15169.545,E2 -15169.545} C_VEL
LIN {X 0,Y 357.125,Z 285.263,A -85,B 0,C 180,E1 -15170.349,E2 -15170.349} C_VEL
LIN {X 0,Y 350.442,Z 434.729,A -85,B 0,C 180,E1 -15173.598,E2 -15173.598} C_VEL
LIN {X 0,Y 348.797,Z 451.83,A -85,B 0,C 180,E1 -15174.156,E2 -15174.156} C_VEL
LIN {X 0,Y 346.801,Z 467.705,A -85,B 0,C 180,E1 -15174.897,E2 -15174.897} C_VEL
LIN {X 0,Y 344.396,Z 483.424,A -85,B 0,C 180,E1 -15175.86,E2 -15175.86} C_VEL
LIN {X 0,Y 341.755,Z 498.027,A -85,B 0,C 180,E1 -15176.976,E2 -15176.976} C_VEL
LIN {X 0,Y 338.9,Z 512.019,A -85,B 0,C 180,E1 -15178.301,E2 -15178.301} C_VEL
LIN {X 0,Y 335.785,Z 525.617,A -85,B 0,C 180,E1 -15179.844,E2 -15179.844} C_VEL
LIN {X 0,Y 332.721,Z 538.608,A -85,B 0,C 180,E1 -15181.621,E2 -15181.621} C_VEL
LIN {X 0,Y 329.822,Z 550.226,A -85,B 0,C 180,E1 -15183.502,E2 -15183.502} C_VEL
LIN {X 0,Y 326.718,Z 562.408,A -85,B 0,C 180,E1 -15185.874,E2 -15185.874} C_VEL
LIN {X 0,Y 324.018,Z 573.004,A -85,B 0,C 180,E1 -15188.36,E2 -15188.36} C_VEL
LIN {X 0,Y 322.03,Z 581.923,A -85,B 0,C 180,E1 -15190.889,E2 -15190.889} C_VEL
LIN {X 0,Y 320.327,Z 589.42,A -85,B 0,C 180,E1 -15193.425,E2 -15193.425} C_VEL
LIN {X 0,Y 319.211,Z 595.596,A -85,B 0,C 180,E1 -15195.982,E2 -15195.982} C_VEL
LIN {X 0,Y 318.394,Z 600.58,A -85,B 0,C 180,E1 -15198.539,E2 -15198.539} C_VEL
LIN {X 0,Y 317.944,Z 604.531,A -85,B 0,C 180,E1 -15201.096,E2 -15201.096} C_VEL
LIN {X 0,Y 317.803,Z 607.995,A -85,B 0,C 180,E1 -15204.347,E2 -15204.347} C_VEL
LIN {X 0,Y 317.756,Z 609.26,A -85,B 0,C 180,E1 -15206.193,E2 -15206.193} C_VEL
LIN {X 0,Y 317.744,Z 610.083,A -85,B 0,C 180,E1 -15208.73,E2 -15208.73} C_VEL
LIN {X 0,Y 317.747,Z 610.017,A -85,B 0,C 180,E1 -15211.264,E2 -15211.264} C_VEL
LIN {X 0,Y 317.771,Z 608.871,A -85,B 0,C 180,E1 -15213.801,E2 -15213.801} C_VEL
LIN {X 0,Y 317.8,Z 606.813,A -85,B 0,C 180,E1 -15216.345,E2 -15216.345} C_VEL
LIN {X 0,Y 317.938,Z 603.625,A -85,B 0,C 180,E1 -15218.898,E2 -15218.898} C_VEL
LIN {X 0,Y 318.367,Z 599.432,A -85,B 0,C 180,E1 -15221.456,E2 -15221.456} C_VEL
LIN {X 0,Y 319.312,Z 593.071,A -85,B 0,C 180,E1 -15224.437,E2 -15224.437} C_VEL
LIN {X 0,Y 320.54,Z 585.558,A -85,B 0,C 180,E1 -15227.213,E2 -15227.213} C_VEL
LIN {X 0,Y 322.017,Z 578.288,A -85,B 0,C 180,E1 -15229.437,E2 -15229.437} C_VEL
LIN {X 0,Y 323.77,Z 569.849,A -85,B 0,C 180,E1 -15231.651,E2 -15231.651} C_VEL
LIN {X 0,Y 326.363,Z 558.388,A -85,B 0,C 180,E1 -15234.147,E2 -15234.147} C_VEL
LIN {X 0,Y 328.733,Z 547.593,A -85,B 0,C 180,E1 -15236.115,E2 -15236.115} C_VEL
LIN {X 0,Y 331.443,Z 535.575,A -85,B 0,C 180,E1 -15237.974,E2 -15237.974} C_VEL
LIN {X 0,Y 334.085,Z 523.007,A -85,B 0,C 180,E1 -15239.623,E2 -15239.623} C_VEL
LIN {X 0,Y 336.787,Z 509.131,A -85,B 0,C 180,E1 -15241.13,E2 -15241.13} C_VEL
LIN {X 0,Y 339.337,Z 494.978,A -85,B 0,C 180,E1 -15242.4,E2 -15242.4} C_VEL
LIN {X 0,Y 341.787,Z 479.309,A -85,B 0,C 180,E1 -15243.542,E2 -15243.542} C_VEL
LIN {X 0,Y 343.86,Z 463.262,A -85,B 0,C 180,E1 -15244.459,E2 -15244.459} C_VEL
LIN {X 0,Y 345.664,Z 446.436,A -85,B 0,C 180,E1 -15245.154,E2 -15245.154} C_VEL
LIN {X 0,Y 346.802,Z 429.442,A -85,B 0,C 180,E1 -15245.634,E2 -15245.634} C_VEL
LIN {X 0,Y 352.438,Z 283.164,A -85,B 0,C 180,E1 -15248.75,E2 -15248.75} C_VEL
LIN {X 0,Y 344.339,Z 266.018,A -85,B 0,C 180,E1 -15250.205,E2 -15250.205} C_VEL
LIN {X 0,Y 333.781,Z 246.001,A -85,B 0,C 180,E1 -15252.17,E2 -15252.17} C_VEL
LIN {X 0,Y 324.923,Z 230.896,A -85,B 0,C 180,E1 -15253.902,E2 -15253.902} C_VEL
LIN {X 0,Y 323.002,Z 227.54,A -85,B 0,C 180,E1 -15254.326,E2 -15254.326} C_VEL
LIN {X 0,Y 319.533,Z 217.99,A -85,B 0,C 180,E1 -15256.734,E2 -15256.734} C_VEL
LIN {X 0,Y 319.56,Z 217.986,A -85,B 0,C 180,E1 -15260.374,E2 -15260.374} C_VEL
LIN {X 0,Y 319.535,Z 217.978,A -85,B 0,C 180,E1 -15263.57,E2 -15263.57} C_VEL
LIN {X 0,Y 319.552,Z 217.983,A -85,B 0,C 180,E1 -15266.684,E2 -15266.684} C_VEL
LIN {X 0,Y 319.558,Z 217.984,A -85,B 0,C 180,E1 -15269.614,E2 -15269.614} C_VEL
LIN {X 0,Y 319.578,Z 217.974,A -85,B 0,C 180,E1 -15272.496,E2 -15272.496} C_VEL
LIN {X 0,Y 319.584,Z 217.977,A -85,B 0,C 180,E1 -15275.303,E2 -15275.303} C_VEL
LIN {X 0,Y 319.604,Z 217.959,A -85,B 0,C 180,E1 -15279.401,E2 -15279.401} C_VEL
LIN {X 0,Y 319.63,Z 217.971,A -85,B 0,C 180,E1 -15282.072,E2 -15282.072} C_VEL
LIN {X 0,Y 319.703,Z 217.952,A -85,B 0,C 180,E1 -15286.007,E2 -15286.007} C_VEL
LIN {X 0,Y 319.729,Z 217.956,A -85,B 0,C 180,E1 -15289.873,E2 -15289.873} C_VEL
LIN {X 0,Y 319.898,Z 217.951,A -85,B 0,C 180,E1 -15292.426,E2 -15292.426} C_VEL
LIN {X 0,Y 319.718,Z 217.939,A -85,B 0,C 180,E1 -15294.956,E2 -15294.956} C_VEL
LIN {X 0,Y 319.961,Z 217.905,A -85,B 0,C 180,E1 -15297.483,E2 -15297.483} C_VEL
LIN {X 0,Y 320.121,Z 217.918,A -85,B 0,C 180,E1 -15300.001,E2 -15300.001} C_VEL
LIN {X 0,Y 319.961,Z 217.933,A -85,B 0,C 180,E1 -15302.518,E2 -15302.518} C_VEL
LIN {X 0,Y 319.888,Z 217.939,A -85,B 0,C 180,E1 -15306.693,E2 -15306.693} C_VEL
LIN {X 0,Y 319.724,Z 217.956,A -85,B 0,C 180,E1 -15310.129,E2 -15310.129} C_VEL
LIN {X 0,Y 319.704,Z 217.972,A -85,B 0,C 180,E1 -15314.726,E2 -15314.726} C_VEL
LIN {X 0,Y 319.663,Z 217.952,A -85,B 0,C 180,E1 -15319.04,E2 -15319.04} C_VEL
LIN {X 0,Y 319.545,Z 217.989,A -85,B 0,C 180,E1 -15323.322,E2 -15323.322} C_VEL
LIN {X 0,Y 319.595,Z 217.962,A -85,B 0,C 180,E1 -15326.092,E2 -15326.092} C_VEL
LIN {X 0,Y 319.567,Z 217.991,A -85,B 0,C 180,E1 -15328.937,E2 -15328.937} C_VEL
LIN {X 0,Y 319.51,Z 217.98,A -85,B 0,C 180,E1 -15331.865,E2 -15331.865} C_VEL
LIN {X 0,Y 319.559,Z 217.99,A -85,B 0,C 180,E1 -15335.546,E2 -15335.546} C_VEL
LIN {X 0,Y 319.541,Z 217.972,A -85,B 0,C 180,E1 -15339.672,E2 -15339.672} C_VEL
LIN {X 0,Y 319.504,Z 217.996,A -85,B 0,C 180,E1 -15343.464,E2 -15343.464} C_VEL
LIN {X 0,Y 319.538,Z 217.993,A -85,B 0,C 180,E1 -15347.02,E2 -15347.02} C_VEL
LIN {X 0,Y 319.532,Z 217.979,A -85,B 0,C 180,E1 -15350.374,E2 -15350.374} C_VEL
LIN {X 0,Y 319.569,Z 217.98,A -85,B 0,C 180,E1 -15354.461,E2 -15354.461} C_VEL
LIN {X 0,Y 319.515,Z 217.999,A -85,B 0,C 180,E1 -15358.141,E2 -15358.141} C_VEL
LIN {X 0,Y 319.564,Z 217.99,A -85,B 0,C 180,E1 -15361.607,E2 -15361.607} C_VEL
LIN {X 0,Y 319.568,Z 217.989,A -85,B 0,C 180,E1 -15365.305,E2 -15365.305} C_VEL
LIN {X 0,Y 319.561,Z 217.984,A -85,B 0,C 180,E1 -15368.049,E2 -15368.049} C_VEL
LIN {X 0,Y 319.605,Z 217.989,A -85,B 0,C 180,E1 -15372.074,E2 -15372.074} C_VEL
LIN {X 0,Y 319.615,Z 218.083,A -85,B 0,C 180,E1 -15372.393,E2 -15372.393} C_VEL
LIN {X 0,Y 320.608,Z 220.838,A -85,B 0,C 180,E1 -15372.635,E2 -15372.635} C_VEL
LIN {X 0,Y 322.511,Z 223.227,A -85,B 0,C 180,E1 -15373.005,E2 -15373.005} C_VEL
LIN {X 0,Y 324.742,Z 226.634,A -85,B 0,C 180,E1 -15373.448,E2 -15373.448} C_VEL
LIN {X 0,Y 333.088,Z 239.532,A -85,B 0,C 180,E1 -15375.051,E2 -15375.051} C_VEL
LIN {X 0,Y 343.066,Z 255.95,A -85,B 0,C 180,E1 -15376.858,E2 -15376.858} C_VEL
LIN {X 0,Y 350.957,Z 271.742,A -85,B 0,C 180,E1 -15378.271,E2 -15378.271} C_VEL
LIN {X 0,Y 352.544,Z 275.25,A -85,B 0,C 180,E1 -15378.554,E2 -15378.554} C_VEL
LIN {X 0,Y 346.824,Z 419.137,A -85,B 0,C 180,E1 -15381.628,E2 -15381.628} C_VEL
LIN {X 0,Y 345.468,Z 436.317,A -85,B 0,C 180,E1 -15382.221,E2 -15382.221} C_VEL
LIN {X 0,Y 343.882,Z 451.483,A -85,B 0,C 180,E1 -15382.96,E2 -15382.96} C_VEL
LIN {X 0,Y 341.842,Z 467.269,A -85,B 0,C 180,E1 -15383.955,E2 -15383.955} C_VEL
LIN {X 0,Y 339.643,Z 481.858,A -85,B 0,C 180,E1 -15385.107,E2 -15385.107} C_VEL
LIN {X 0,Y 336.948,Z 496.923,A -85,B 0,C 180,E1 -15386.565,E2 -15386.565} C_VEL
LIN {X 0,Y 334.229,Z 510.688,A -85,B 0,C 180,E1 -15388.195,E2 -15388.195} C_VEL
LIN {X 0,Y 331.436,Z 523.489,A -85,B 0,C 180,E1 -15390.003,E2 -15390.003} C_VEL
LIN {X 0,Y 328.619,Z 536.142,A -85,B 0,C 180,E1 -15392.148,E2 -15392.148} C_VEL
LIN {X 0,Y 326.124,Z 546.94,A -85,B 0,C 180,E1 -15394.328,E2 -15394.328} C_VEL
LIN {X 0,Y 323.994,Z 556.158,A -85,B 0,C 180,E1 -15396.542,E2 -15396.542} C_VEL
LIN {X 0,Y 322.027,Z 565.054,A -85,B 0,C 180,E1 -15399.107,E2 -15399.107} C_VEL
LIN {X 0,Y 320.659,Z 571.658,A -85,B 0,C 180,E1 -15401.379,E2 -15401.379} C_VEL
LIN {X 0,Y 319.471,Z 577.945,A -85,B 0,C 180,E1 -15404.006,E2 -15404.006} C_VEL
LIN {X 0,Y 318.633,Z 582.971,A -85,B 0,C 180,E1 -15406.665,E2 -15406.665} C_VEL
LIN {X 0,Y 318.05,Z 586.899,A -85,B 0,C 180,E1 -15409.36,E2 -15409.36} C_VEL
LIN {X 0,Y 317.621,Z 589.693,A -85,B 0,C 180,E1 -15412.098,E2 -15412.098} C_VEL
LIN {X 0,Y 317.439,Z 591.332,A -85,B 0,C 180,E1 -15414.878,E2 -15414.878} C_VEL
LIN {X 0,Y 317.477,Z 591.866,A -85,B 0,C 180,E1 -15417.705,E2 -15417.705} C_VEL
LIN {X 0,Y 317.571,Z 591.177,A -85,B 0,C 180,E1 -15420.599,E2 -15420.599} C_VEL
LIN {X 0,Y 317.891,Z 589.156,A -85,B 0,C 180,E1 -15423.555,E2 -15423.555} C_VEL
LIN {X 0,Y 318.168,Z 587.528,A -85,B 0,C 180,E1 -15425.151,E2 -15425.151} C_VEL
LIN {X 0,Y 317.72,Z 586.348,A -85,B 0,C 180,E1 -15426.189,E2 -15426.189} C_VEL
LIN {X 0,Y 315.315,Z 584.173,A -85,B 0,C 180,E1 -15427.886,E2 -15427.886} C_VEL
LIN {X 0,Y 313.369,Z 582.213,A -85,B 0,C 180,E1 -15429.246,E2 -15429.246} C_VEL
LIN {X 0,Y 312.761,Z 580.433,A -85,B 0,C 180,E1 -15430.278,E2 -15430.278} C_VEL
LIN {X 0,Y 312.836,Z 579.795,A -85,B 0,C 180,E1 -15430.621,E2 -15430.621} C_VEL
LIN {X 0,Y 314.023,Z 574.586,A -85,B 0,C 180,E1 -15433.049,E2 -15433.049} C_VEL
LIN {X 0,Y 315.997,Z 566.855,A -85,B 0,C 180,E1 -15435.965,E2 -15435.965} C_VEL
LIN {X 0,Y 318.452,Z 558.138,A -85,B 0,C 180,E1 -15438.623,E2 -15438.623} C_VEL
LIN {X 0,Y 321.11,Z 548.348,A -85,B 0,C 180,E1 -15441.089,E2 -15441.089} C_VEL
LIN {X 0,Y 324.092,Z 537.545,A -85,B 0,C 180,E1 -15443.357,E2 -15443.357} C_VEL
LIN {X 0,Y 327.344,Z 525.44,A -85,B 0,C 180,E1 -15445.479,E2 -15445.479} C_VEL
LIN {X 0,Y 330.631,Z 512.423,A -85,B 0,C 180,E1 -15447.384,E2 -15447.384} C_VEL
LIN {X 0,Y 333.806,Z 498.875,A -85,B 0,C 180,E1 -15449.031,E2 -15449.031} C_VEL
LIN {X 0,Y 337.083,Z 483.02,A -85,B 0,C 180,E1 -15450.604,E2 -15450.604} C_VEL
LIN {X 0,Y 339.675,Z 468.647,A -85,B 0,C 180,E1 -15451.747,E2 -15451.747} C_VEL
LIN {X 0,Y 341.962,Z 453.392,A -85,B 0,C 180,E1 -15452.727,E2 -15452.727} C_VEL
LIN {X 0,Y 343.902,Z 437.49,A -85,B 0,C 180,E1 -15453.511,E2 -15453.511} C_VEL
LIN {X 0,Y 345.191,Z 422.834,A -85,B 0,C 180,E1 -15454.039,E2 -15454.039} C_VEL
LIN {X 0,Y 346.422,Z 398.96,A -85,B 0,C 180,E1 -15454.616,E2 -15454.616} C_VEL
LIN {X 0,Y 352.028,Z 280.315,A -85,B 0,C 180,E1 -15457.208,E2 -15457.208} C_VEL
LIN {X 0,Y 345.244,Z 267.022,A -85,B 0,C 180,E1 -15458.714,E2 -15458.714} C_VEL
LIN {X 0,Y 339.488,Z 256.967,A -85,B 0,C 180,E1 -15460.052,E2 -15460.052} C_VEL
LIN {X 0,Y 332.034,Z 245.735,A -85,B 0,C 180,E1 -15461.878,E2 -15461.878} C_VEL
LIN {X 0,Y 326.27,Z 237.582,A -85,B 0,C 180,E1 -15463.396,E2 -15463.396} C_VEL
LIN {X 0,Y 323.202,Z 233.488,A -85,B 0,C 180,E1 -15464.247,E2 -15464.247} C_VEL
LIN {X 0,Y 320.546,Z 229.813,A -85,B 0,C 180,E1 -15465.025,E2 -15465.025} C_VEL
LIN {X 0,Y 317.457,Z 226.137,A -85,B 0,C 180,E1 -15465.946,E2 -15465.946} C_VEL
LIN {X 0,Y 316.499,Z 224.3,A -85,B 0,C 180,E1 -15466.271,E2 -15466.271} C_VEL
LIN {X 0,Y 314.13,Z 222.363,A -85,B 0,C 180,E1 -15466.989,E2 -15466.989} C_VEL
LIN {X 0,Y 312.896,Z 220.03,A -85,B 0,C 180,E1 -15467.432,E2 -15467.432} C_VEL
LIN {X 0,Y 312.634,Z 218.852,A -85,B 0,C 180,E1 -15467.586,E2 -15467.586} C_VEL
LIN {X 0,Y 312.795,Z 218.831,A -85,B 0,C 180,E1 -15471.349,E2 -15471.349} C_VEL
LIN {X 0,Y 312.903,Z 218.818,A -85,B 0,C 180,E1 -15473.551,E2 -15473.551} C_VEL
LIN {X 0,Y 312.937,Z 218.816,A -85,B 0,C 180,E1 -15477.425,E2 -15477.425} C_VEL
LIN {X 0,Y 313.071,Z 218.799,A -85,B 0,C 180,E1 -15479.999,E2 -15479.999} C_VEL
LIN {X 0,Y 312.936,Z 218.815,A -85,B 0,C 180,E1 -15482.574,E2 -15482.574} C_VEL
LIN {X 0,Y 312.859,Z 218.826,A -85,B 0,C 180,E1 -15486.448,E2 -15486.448} C_VEL
LIN {X 0,Y 312.755,Z 218.841,A -85,B 0,C 180,E1 -15489.049,E2 -15489.049} C_VEL
LIN {X 0,Y 312.635,Z 218.848,A -85,B 0,C 180,E1 -15492.99,E2 -15492.99} C_VEL
LIN {X 0,Y 312.625,Z 218.85,A -85,B 0,C 180,E1 -15495.65,E2 -15495.65} C_VEL
LIN {X 0,Y 312.542,Z 218.863,A -85,B 0,C 180,E1 -15499.712,E2 -15499.712} C_VEL
LIN {X 0,Y 312.53,Z 218.866,A -85,B 0,C 180,E1 -15502.779,E2 -15502.779} C_VEL
LIN {X 0,Y 312.606,Z 218.858,A -85,B 0,C 180,E1 -15505.934,E2 -15505.934} C_VEL
LIN {X 0,Y 312.53,Z 218.862,A -85,B 0,C 180,E1 -15509.651,E2 -15509.651} C_VEL
LIN {X 0,Y 312.523,Z 218.866,A -85,B 0,C 180,E1 -15513.687,E2 -15513.687} C_VEL
LIN {X 0,Y 312.529,Z 218.87,A -85,B 0,C 180,E1 -15517.53,E2 -15517.53} C_VEL
LIN {X 0,Y 312.541,Z 218.983,A -85,B 0,C 180,E1 -15517.674,E2 -15517.674} C_VEL
LIN {X 0,Y 313.732,Z 222.034,A -85,B 0,C 180,E1 -15518.846,E2 -15518.846} C_VEL
LIN {X 0,Y 315.343,Z 225.55,A -85,B 0,C 180,E1 -15520.111,E2 -15520.111} C_VEL
LIN {X 0,Y 319.871,Z 231.745,A -85,B 0,C 180,E1 -15521.522,E2 -15521.522} C_VEL
LIN {X 0,Y 325.921,Z 240.678,A -85,B 0,C 180,E1 -15523.277,E2 -15523.277} C_VEL
LIN {X 0,Y 331.244,Z 248.829,A -85,B 0,C 180,E1 -15524.706,E2 -15524.706} C_VEL
LIN {X 0,Y 338.399,Z 260.856,A -85,B 0,C 180,E1 -15526.509,E2 -15526.509} C_VEL
LIN {X 0,Y 345.689,Z 274.635,A -85,B 0,C 180,E1 -15528.232,E2 -15528.232} C_VEL
LIN {X 0,Y 351.825,Z 287.674,A -85,B 0,C 180,E1 -15529.613,E2 -15529.613} C_VEL
LIN {X 0,Y 344.901,Z 435.29,A -85,B 0,C 180,E1 -15532.872,E2 -15532.872} C_VEL
LIN {X 0,Y 343.188,Z 452.379,A -85,B 0,C 180,E1 -15533.445,E2 -15533.445} C_VEL
LIN {X 0,Y 341.058,Z 468.478,A -85,B 0,C 180,E1 -15534.216,E2 -15534.216} C_VEL
LIN {X 0,Y 338.566,Z 483.965,A -85,B 0,C 180,E1 -15535.189,E2 -15535.189} C_VEL
LIN {X 0,Y 335.837,Z 498.395,A -85,B 0,C 180,E1 -15536.318,E2 -15536.318} C_VEL
LIN {X 0,Y 332.794,Z 512.625,A -85,B 0,C 180,E1 -15537.691,E2 -15537.691} C_VEL
LIN {X 0,Y 329.36,Z 526.952,A -85,B 0,C 180,E1 -15539.37,E2 -15539.37} C_VEL
LIN {X 0,Y 326.445,Z 538.707,A -85,B 0,C 180,E1 -15541.025,E2 -15541.025} C_VEL
LIN {X 0,Y 323.244,Z 550.923,A -85,B 0,C 180,E1 -15543.052,E2 -15543.052} C_VEL
LIN {X 0,Y 320.163,Z 562.439,A -85,B 0,C 180,E1 -15545.348,E2 -15545.348} C_VEL
LIN {X 0,Y 317.325,Z 572.975,A -85,B 0,C 180,E1 -15547.88,E2 -15547.88} C_VEL
LIN {X 0,Y 315.196,Z 581.849,A -85,B 0,C 180,E1 -15550.458,E2 -15550.458} C_VEL
LIN {X 0,Y 313.425,Z 589.319,A -85,B 0,C 180,E1 -15553.05,E2 -15553.05} C_VEL
LIN {X 0,Y 312.234,Z 595.486,A -85,B 0,C 180,E1 -15555.662,E2 -15555.662} C_VEL
LIN {X 0,Y 311.384,Z 600.446,A -85,B 0,C 180,E1 -15558.277,E2 -15558.277} C_VEL
LIN {X 0,Y 310.874,Z 604.381,A -85,B 0,C 180,E1 -15560.892,E2 -15560.892} C_VEL
LIN {X 0,Y 310.722,Z 607.964,A -85,B 0,C 180,E1 -15564.381,E2 -15564.381} C_VEL
LIN {X 0,Y 310.673,Z 609.591,A -85,B 0,C 180,E1 -15567.404,E2 -15567.404} C_VEL
LIN {X 0,Y 310.689,Z 609.957,A -85,B 0,C 180,E1 -15569.997,E2 -15569.997} C_VEL
LIN {X 0,Y 310.681,Z 609.336,A -85,B 0,C 180,E1 -15572.59,E2 -15572.59} C_VEL
LIN {X 0,Y 310.718,Z 607.347,A -85,B 0,C 180,E1 -15575.612,E2 -15575.612} C_VEL
LIN {X 0,Y 310.769,Z 605.09,A -85,B 0,C 180,E1 -15577.795,E2 -15577.795} C_VEL
LIN {X 0,Y 311.185,Z 600.293,A -85,B 0,C 180,E1 -15581.064,E2 -15581.064} C_VEL
LIN {X 0,Y 311.949,Z 595.183,A -85,B 0,C 180,E1 -15583.68,E2 -15583.68} C_VEL
LIN {X 0,Y 312.964,Z 588.9,A -85,B 0,C 180,E1 -15586.298,E2 -15586.298} C_VEL
LIN {X 0,Y 314.768,Z 580.153,A -85,B 0,C 180,E1 -15589.224,E2 -15589.224} C_VEL
LIN {X 0,Y 316.767,Z 570.694,A -85,B 0,C 180,E1 -15591.811,E2 -15591.811} C_VEL
LIN {X 0,Y 319.036,Z 560.941,A -85,B 0,C 180,E1 -15594.046,E2 -15594.046} C_VEL
LIN {X 0,Y 321.749,Z 549.25,A -85,B 0,C 180,E1 -15596.306,E2 -15596.306} C_VEL
LIN {X 0,Y 324.586,Z 537.149,A -85,B 0,C 180,E1 -15598.266,E2 -15598.266} C_VEL
LIN {X 0,Y 327.575,Z 523.57,A -85,B 0,C 180,E1 -15600.095,E2 -15600.095} C_VEL
LIN {X 0,Y 330.401,Z 509.633,A -85,B 0,C 180,E1 -15601.65,E2 -15601.65} C_VEL
LIN {X 0,Y 332.974,Z 495.918,A -85,B 0,C 180,E1 -15602.917,E2 -15602.917} C_VEL
LIN {X 0,Y 335.49,Z 480.56,A -85,B 0,C 180,E1 -15604.076,E2 -15604.076} C_VEL
LIN {X 0,Y 337.649,Z 464.827,A -85,B 0,C 180,E1 -15605.004,E2 -15605.004} C_VEL
LIN {X 0,Y 339.466,Z 448.512,A -85,B 0,C 180,E1 -15605.715,E2 -15605.715} C_VEL
LIN {X 0,Y 340.704,Z 432.857,A -85,B 0,C 180,E1 -15606.196,E2 -15606.196} C_VEL
LIN {X 0,Y 346.683,Z 285.444,A -85,B 0,C 180,E1 -15609.388,E2 -15609.388} C_VEL
LIN {X 0,Y 338.142,Z 267.54,A -85,B 0,C 180,E1 -15610.964,E2 -15610.964} C_VEL
LIN {X 0,Y 329.226,Z 250.587,A -85,B 0,C 180,E1 -15612.682,E2 -15612.682} C_VEL
LIN {X 0,Y 320.287,Z 235.225,A -85,B 0,C 180,E1 -15614.48,E2 -15614.48} C_VEL
LIN {X 0,Y 315.606,Z 227.438,A -85,B 0,C 180,E1 -15615.474,E2 -15615.474} C_VEL
LIN {X 0,Y 312.48,Z 218.874,A -85,B 0,C 180,E1 -15617.736,E2 -15617.736} C_VEL
LIN {X 0,Y 312.52,Z 218.864,A -85,B 0,C 180,E1 -15621.906,E2 -15621.906} C_VEL
LIN {X 0,Y 312.482,Z 218.874,A -85,B 0,C 180,E1 -15625.788,E2 -15625.788} C_VEL
LIN {X 0,Y 312.493,Z 218.853,A -85,B 0,C 180,E1 -15628.851,E2 -15628.851} C_VEL
LIN {X 0,Y 312.543,Z 218.862,A -85,B 0,C 180,E1 -15631.822,E2 -15631.822} C_VEL
LIN {X 0,Y 312.561,Z 218.843,A -85,B 0,C 180,E1 -15634.709,E2 -15634.709} C_VEL
LIN {X 0,Y 312.566,Z 218.862,A -85,B 0,C 180,E1 -15637.528,E2 -15637.528} C_VEL
LIN {X 0,Y 312.611,Z 218.836,A -85,B 0,C 180,E1 -15641.655,E2 -15641.655} C_VEL
LIN {X 0,Y 312.665,Z 218.835,A -85,B 0,C 180,E1 -15645.686,E2 -15645.686} C_VEL
LIN {X 0,Y 312.674,Z 218.828,A -85,B 0,C 180,E1 -15649.642,E2 -15649.642} C_VEL
LIN {X 0,Y 312.838,Z 218.83,A -85,B 0,C 180,E1 -15652.254,E2 -15652.254} C_VEL
LIN {X 0,Y 312.688,Z 218.816,A -85,B 0,C 180,E1 -15654.843,E2 -15654.843} C_VEL
LIN {X 0,Y 312.963,Z 218.794,A -85,B 0,C 180,E1 -15658.714,E2 -15658.714} C_VEL
LIN {X 0,Y 312.962,Z 218.812,A -85,B 0,C 180,E1 -15661.287,E2 -15661.287} C_VEL
LIN {X 0,Y 312.686,Z 218.824,A -85,B 0,C 180,E1 -15665.159,E2 -15665.159} C_VEL
LIN {X 0,Y 312.825,Z 218.828,A -85,B 0,C 180,E1 -15667.748,E2 -15667.748} C_VEL
LIN {X 0,Y 312.64,Z 218.823,A -85,B 0,C 180,E1 -15671.673,E2 -15671.673} C_VEL
LIN {X 0,Y 312.673,Z 218.849,A -85,B 0,C 180,E1 -15674.889,E2 -15674.889} C_VEL
LIN {X 0,Y 312.605,Z 218.831,A -85,B 0,C 180,E1 -15679.239,E2 -15679.239} C_VEL
LIN {X 0,Y 312.521,Z 218.867,A -85,B 0,C 180,E1 -15682.791,E2 -15682.791} C_VEL
LIN {X 0,Y 312.573,Z 218.836,A -85,B 0,C 180,E1 -15685.936,E2 -15685.936} C_VEL
LIN {X 0,Y 312.523,Z 218.868,A -85,B 0,C 180,E1 -15689.653,E2 -15689.653} C_VEL
